# B&R Automation Studio project NAINV104C00R8L515F00 (part 35)

### Program Logical/LCS/LCSLF (IEC) - 1.00.0 - NtRecipe v5.00.0 , NtFileIO v5.00.0

#### InputRef.var
```iecst
(*2019-06-28*)
(**)
(*General*)
VAR
	p_eAct : REFERENCE TO eLCSAction;
	p_udiRstErr : REFERENCE TO UDINT;
	p_bPrep : REFERENCE TO BOOL;
	p_bEn : REFERENCE TO BOOL;
	p_bDis : REFERENCE TO BOOL;
END_VAR
(**)
(*Configuration*)
VAR
	p_tyCurrProdParam : REFERENCE TO tyProdRcpParam;
	p_bMnlAccData : REFERENCE TO BOOL;
	p_bAccData : REFERENCE TO BOOL;
	p_tyLCSProdRcpInfo : REFERENCE TO tyProdRcpParam;
	p_bChkLmtOK : REFERENCE TO BOOL;
	p_bChkLmtNG : REFERENCE TO BOOL;
	p_bAccNewRcpCond : REFERENCE TO BOOL;
	p_bUpdtNewRcpCond : REFERENCE TO BOOL;
	p_bAutoUpdtData : REFERENCE TO BOOL;
	p_bUIUpdtData : REFERENCE TO BOOL;
	p_sInfoMsg : REFERENCE TO STRING[200];
	p_sProgNm : REFERENCE TO STRING[15];
	p_bNtSettingsLoadDone : REFERENCE TO BOOL;
	p_bUIBtnSectionLdr : REFERENCE TO BOOL;
	p_bLCSSectionLeaderEn : REFERENCE TO BOOL;
	p_bMcParamSectionLdr : REFERENCE TO BOOL;
END_VAR
```

#### InputRef_Link.var
```iecst
(*2019-04-24*)
(**)
VAR
	sWidthInUMTemp : STRING[80];
	p_bLinkStartupRun : REFERENCE TO BOOL;
	p_eLinkMcParamUSCommMod : REFERENCE TO eMcSetCommMod;
END_VAR
(**)
VAR
	p_bLinkOpsRun : REFERENCE TO BOOL;
	p_bLinkMcParam : REFERENCE TO tyMcParam;
	p_bLinkConvHvBrd : REFERENCE TO BOOL;
END_VAR
```

#### Local.var
```iecst
(*2019-06-28*)
(**)
(*Local Action, State & Status*)
VAR
	eAct : eLCSAction := LCSActIdle;
	eStat : eLCSAction := LCSActIdle;
	eStatus : eFBStatus := Idle;
	udiStatus : UDINT := 0;
	sStatTxt : STRING[200] := '';
	a_sStatText : ARRAY[0..50] OF STRING[200] := ['Idling','Adding Product','Adding Multiple Products','Editing Product','Editing Multiple Products','OverWrite Product','OverWrite Multiple Products','Deleting Product','Deleting Multiple Products','Running LCS Product','Uploading Product','Uploading Multiple Products',39('')];
END_VAR
(**)
(*Local Alarm*)
VAR
	tyAlmData : tyAlmDat;
	tyInfoData : tyAlmDat;
	a_tyAlmText : ARRAY[10000..10099] OF tyAlmTxt;
END_VAR
(**)
(*Local Output*)
VAR
	udiPLCStatus : UDINT;
	bChkLmt : BOOL;
	bAccDataMnl : BOOL;
	bUpdtDataMnl : BOOL;
	sUpdtProdRcpNm : STRING[30];
	diUpdtProdWidth : DINT;
END_VAR
(**)
(*Local Input*)
VAR
	udiRstErr : UDINT := 0;
	bPrep : BOOL := TRUE;
	bEn : BOOL := TRUE;
	bDis : BOOL := FALSE;
	tyCurrProdParam : tyProdRcpParam;
	bMnlAccData : BOOL;
	bAccData : BOOL;
	tyLCSProdRcpInfo : tyProdRcpParam;
	bChkLmtOK : BOOL;
	bChkLmtNG : BOOL;
	bAccNewRcpCond : BOOL;
	bUpdtNewRcpCond : BOOL;
	bAutoUpdtData : BOOL;
	bUIUpdtData : BOOL;
	sInfoMsg : STRING[200];
	sProgNm : STRING[15] := 'LCSLF';
	bNtSettingsLoadDone : BOOL := TRUE;
END_VAR
(**)
(*Local*)
VAR
	bRstErr : BOOL;
	udiRstErrOld : UDINT;
	bInitDone : BOOL;
	bInitialDone : BOOL;
	usiStep : USINT;
	usiProdUpdtDatStep : USINT;
	udiModuleNum : UDINT := 4101;
END_VAR
```

#### Act_Action.st
```iecst
(** 2019-04-24 **)
ACTION Act_Action:

	//Reset Error
	IF (eStatus = Error) AND bRstErr THEN
		p_eAct	:= LCSActIdle;
		eStat	:= LCSActIdle;
	END_IF

	//Reset Done
	IF eStatus = Done AND p_eAct = LCSActIdle THEN
		eStat	:= LCSActIdle;
	END_IF

	//Set p_eAct
	IF eStatus = Idle THEN
		eStat	:= p_eAct;
	END_IF

END_ACTION
```

#### Act_Alarm.st
```iecst
(** 2019-04-24 **)
ACTION Act_Alarm:

	//Error
	IF EDGEPOS(eStatus = Error) THEN

		tyAlmData.sProgNm		:= p_sProgNm;
		tyAlmData.udiCode		:= udiStatus;
		tyAlmData.eSeverity		:= AlmSeverityError;
		tyAlmData.udiRunTime	:= tyAlmData.udiRunTime + 1;
		tyAlmData.bAlm			:= TRUE;
		tyAlmData.udiModuleNum  := udiModuleNum;
		g_sLCSLFProgNm			:= p_sProgNm;

		//Get Error Message
		IF tyAlmData.udiCode < 10000 OR tyAlmData.udiCode > 10099 THEN
			tyAlmData.sAlmMsg	:= 'Unknown';
			tyAlmData.sRcyMsg	:= 'Unknown';
		ELSE
			tyAlmData.sAlmMsg	:= a_tyAlmText[tyAlmData.udiCode].sAlmText;
			tyAlmData.sRcyMsg	:= a_tyAlmText[tyAlmData.udiCode].sRcyText;
		END_IF

		sStatTxt	:= tyAlmData.sAlmMsg;

	ELSIF bRstErr AND (tyAlmData.udiCode <> 0) THEN

		tyAlmData.udiCode	:= 0;
		tyAlmData.eSeverity	:= AlmSeverityNA;
		tyAlmData.sAlmMsg	:= '';
		tyAlmData.sRcyMsg	:= '';
		tyAlmData.bAlm			:= FALSE;
		sStatTxt	:= a_sStatText[eStat];

	END_IF

END_ACTION
```

#### Act_Background.st
```iecst
(** 2019-06-12 **)
ACTION Act_Background:

	//Update To Leader Recipe
	CASE usiProdUpdtDatStep OF
		0:
			//Update New Recipe Condition
			IF sUpdtProdRcpNm <> '' THEN
				IF (p_tyCurrProdParam.sRcpNm <> sUpdtProdRcpNm) THEN
					IF p_bUpdtNewRcpCond = TRUE THEN
						usiProdUpdtDatStep	:= 1;
					END_IF
				END_IF
			ELSE
				sUpdtProdRcpNm	:= p_tyCurrProdParam.sRcpNm;
				diUpdtProdWidth	:= p_tyCurrProdParam.diWidthInUM;
			END_IF

		1:
			//Manual Update Data Check
			IF p_bAutoUpdtData = FALSE THEN
				bUpdtDataMnl	:= TRUE;

				IF p_bUIUpdtData = TRUE THEN
					bUpdtDataMnl	:= FALSE;
					usiProdUpdtDatStep	:= 2;
				END_IF
			ELSE
				bUpdtDataMnl	:= FALSE;
				usiProdUpdtDatStep	:= 2;
			END_IF

		2:
			//Update New Recipe
			sUpdtProdRcpNm	:= p_tyCurrProdParam.sRcpNm;
			diUpdtProdWidth	:= p_tyCurrProdParam.diWidthInUM;

			usiProdUpdtDatStep	:= 0;

	END_CASE

END_ACTION
```

#### Act_InitGlobal.st
```iecst
(** 2019-05-07 **)
ACTION Act_InitGlobal:

	(* Always Change If Project Change *)

	//Pass Data To Link
	p_bLinkStartupRun ACCESS p_StartupRun;
	p_eLinkMcParamUSCommMod ACCESS p_McParamUSCommMod;
	p_bLinkConvHvBrd ACCESS p_OpsInvertHvBrd;

	p_bLinkOpsRun ACCESS p_OpsRun;

	//Pass Data To Internal Use
	p_eAct ACCESS p_LCS_LCSLF_LCSAct;
	p_udiRstErr ACCESS p_RstErrReset;
	p_bPrep ACCESS p_NtParamLCSLFPrep;
	p_bEn ACCESS p_McParamLCSLFEn;
	p_tyCurrProdParam ACCESS p_ProdRcpCurrRcp0;
	p_bMnlAccData ACCESS p_McParamMnlAccDat;
	p_bAccData ACCESS p_UIProdAccData;
	p_tyLCSProdRcpInfo ACCESS p_LCS_LCSLF_LCSProdRcpInfo;
	p_bChkLmtOK ACCESS p_LCSChkLmtOK;
	p_bChkLmtNG ACCESS p_LCSChkLmtNG;
	p_sProgNm ACCESS p_NtParamLCSLFProgNm;
	p_bNtSettingsLoadDone ACCESS p_StartupNtSettingsLoadDone;

	p_bUIBtnSectionLdr ACCESS P_UISectionLdr;
	p_bLCSSectionLeaderEn ACCESS p_LCSSectionLeaderEn;
	p_bMcParamSectionLdr ACCESS p_McParamSectionLeader;

	(* Always Change If Project Change *)

END_ACTION
```

#### Act_InitLocal.st
```iecst
(** 2019-06-28 **)
ACTION Act_InitLocal:

	//Input Reference Link To Local Variable
	p_eAct ACCESS ADR(eAct);
	p_udiRstErr ACCESS ADR(udiRstErr);
	p_bPrep ACCESS ADR(bPrep);
	p_bEn ACCESS ADR(bEn);
	p_bDis ACCESS ADR(bDis);
	p_tyCurrProdParam ACCESS ADR(tyCurrProdParam);
	p_bMnlAccData ACCESS ADR(bMnlAccData);
	p_bAccData ACCESS ADR(bAccData);
	p_tyLCSProdRcpInfo ACCESS ADR(tyLCSProdRcpInfo);
	p_bChkLmtOK ACCESS ADR(bChkLmtOK);
	p_bChkLmtNG ACCESS ADR(bChkLmtNG);
	p_bAccNewRcpCond ACCESS ADR(bAccNewRcpCond);
	p_bUpdtNewRcpCond ACCESS ADR(bUpdtNewRcpCond);
	p_bAutoUpdtData ACCESS ADR(bAutoUpdtData);
	p_bUIUpdtData ACCESS ADR(bUIUpdtData);
	p_sInfoMsg ACCESS ADR(sInfoMsg);
	p_sProgNm ACCESS ADR(sProgNm);
	p_bNtSettingsLoadDone ACCESS ADR(bNtSettingsLoadDone);

END_ACTION
```

#### Act_Link.st
```iecst
(** 2019-06-28 **)
ACTION Act_Link:

	p_sInfoMsg		:= 'LCS Request New Recipe';
	p_sInfoMsg		:= CONCAT(p_sInfoMsg , '$r$n');
	p_sInfoMsg		:= CONCAT(p_sInfoMsg , 'Old Recipe Name : ');
	p_sInfoMsg		:= CONCAT(p_sInfoMsg , p_tyCurrProdParam.sRcpNm);
	p_sInfoMsg		:= CONCAT(p_sInfoMsg , '$r$n');
	p_sInfoMsg		:= CONCAT(p_sInfoMsg , 'Old Recipe Width : ');
	sWidthInUMTemp	:= DINT_TO_STRING(p_tyCurrProdParam.diWidthInUM / 1000);
	p_sInfoMsg		:= CONCAT(p_sInfoMsg , sWidthInUMTemp);
	p_sInfoMsg		:= CONCAT(p_sInfoMsg , '$r$n');
	p_sInfoMsg		:= CONCAT(p_sInfoMsg , 'New Recipe Name : ');
	p_sInfoMsg		:= CONCAT(p_sInfoMsg , p_tyLCSProdRcpInfo.sRcpNm);
	p_sInfoMsg		:= CONCAT(p_sInfoMsg , '$r$n');
	p_sInfoMsg		:= CONCAT(p_sInfoMsg , 'New Recipe Width : ');
	sWidthInUMTemp	:= DINT_TO_STRING(p_tyLCSProdRcpInfo.diWidthInUM / 1000);
	p_sInfoMsg		:= CONCAT(p_sInfoMsg , sWidthInUMTemp);

	//Accept New Recipe Condition
	p_bAccNewRcpCond	:= p_bLinkOpsRun = TRUE AND p_bLinkConvHvBrd = FALSE;

END_ACTION
```

#### Act_LinkAction.st
```iecst
(** 2019-04-24 **)
ACTION Act_LinkAction:

END_ACTION
```

#### Act_LinkEn.st
```iecst
(** 2019-04-24 **)
ACTION Act_LinkEn:

	//Link bPrep, bEn & bDis
	p_bDis	:= (p_bLinkStartupRun = TRUE) OR (p_eLinkMcParamUSCommMod = McSetCommModHermes);

END_ACTION
```

#### Act_Main.st
```iecst
(** 2019-06-28 **)
ACTION Act_Main:

	//Main
	CASE eStat OF

		LCSActIdle:
			IF eStatus <> Idle THEN	//Reset Data
				//Private
				usiStep		:= 0;
				bAccDataMnl	:= FALSE;
				bChkLmt		:= FALSE;

				tyInfoData.sProgNm		:= '';
				tyInfoData.udiCode		:= 0;
				tyInfoData.eSeverity	:= AlmSeverityNA;
				tyInfoData.sAlmMsg		:= '';

				sStatTxt	:= a_sStatText[eStat];

			END_IF

			eStatus			:= Idle;
			udiPLCStatus	:= 65534;

		LCSActRunProd:
			IF eStatus = Idle OR eStatus = Busy THEN

				eStatus			:= Busy;
				udiPLCStatus	:= 65535;

				sStatTxt	:= a_sStatText[eStat];

				CASE usiStep OF
					0:
						//Check Limit
						bChkLmt	:= TRUE;

						IF p_bChkLmtOK = TRUE THEN
							usiStep			:= 1;
						ELSIF p_bChkLmtNG = TRUE THEN
							eStatus			:= Done;
							udiPLCStatus	:= 10010;	//Out Of Range While Accepting New Recipe
						END_IF

					1:
						//Manual Accept Data Check
						IF p_bMnlAccData = TRUE THEN
							bAccDataMnl	:= TRUE;

							//Info Message
							tyInfoData.sProgNm		:= p_sProgNm;
							tyInfoData.udiCode		:= 10000;
							tyInfoData.eSeverity	:= AlmSeverityInfo;
							tyInfoData.sAlmMsg		:= p_sInfoMsg;

							IF p_bAccData = TRUE THEN
								p_bAccData 	:= FALSE; // 2023_07_06_Debug for Manual Accept Data automatically accept after product change many times
								bAccDataMnl	:= FALSE;
								usiStep		:= 2;
							END_IF
						ELSE
							bAccDataMnl	:= FALSE;
							p_bAccData	:= FALSE; // 2023_07_06_Debug for Manual Accept Data automatically accept after product change many times
							usiStep		:= 2;
						END_IF

					2:
						//Accept New Recipe Condition
						IF p_bAccNewRcpCond = TRUE THEN
							usiStep	:= 3;
						ELSE
							//Info Message
							tyInfoData.sProgNm		:= p_sProgNm;
							tyInfoData.udiCode		:= 10000;
							tyInfoData.eSeverity	:= AlmSeverityInfo;
							tyInfoData.sAlmMsg		:= p_sInfoMsg;
						END_IF

					3:
						//Accept New Recipe
						p_tyCurrProdParam	:= p_tyLCSProdRcpInfo;

						IF p_bLCSSectionLeaderEn = TRUE THEN
							p_bMcParamSectionLdr	:= TRUE;
							p_bUIBtnSectionLdr		:= TRUE;
						ELSE
							p_bMcParamSectionLdr	:= FALSE;
							p_bUIBtnSectionLdr		:= FALSE;

						END_IF

						usiStep	:= 4;

					4:
						//Clear Info Message
						tyInfoData.sProgNm		:= '';
						tyInfoData.udiCode		:= 0;
						tyInfoData.eSeverity	:= AlmSeverityNA;
						tyInfoData.sAlmMsg		:= '';

						usiStep	:= 0;

						eStatus			:= Done;
						udiPLCStatus	:= 0;

				END_CASE

			END_IF

		ELSE
			IF eStatus = Idle OR eStatus = Busy THEN
				eStatus	:= Done;
			END_IF

	END_CASE

END_ACTION
```

#### Act_Main_Disable.st
```iecst
(** 2019-06-12 **)
ACTION Act_Main_Disable:

	usiProdUpdtDatStep		:= 0;

END_ACTION
```

#### Act_RstErr.st
```iecst
(** 2019-04-24 **)
ACTION Act_RstErr:

	IF p_udiRstErr <> udiRstErrOld THEN
		bRstErr			:= TRUE;
		udiRstErrOld	:= p_udiRstErr;
	ELSE
		bRstErr			:= FALSE;
	END_IF

END_ACTION
```

#### Cyclic.st
```iecst
(** 2019-04-24 **)
PROGRAM _CYCLIC

	IF bInitDone = FALSE THEN
		bInitDone	:= TRUE;

		Act_InitLocal;
		Act_InitGlobal;

	ELSIF bInitialDone = FALSE THEN
		IF p_bNtSettingsLoadDone = TRUE THEN
			bInitialDone	:= TRUE;

			Act_Initial;
		END_IF

	ELSE

		Act_RstErr;
		Act_LinkAction;
		Act_Action;
		Act_LinkEn;

		IF (p_bPrep = TRUE) AND (p_bEn = TRUE) AND (p_bDis = FALSE) THEN
			Act_Link;
			Act_Background;
			Act_Main;

		ELSE
			Act_Main_Disable;

			IF eStat <> LCSActIdle THEN
				eStatus			:= Done;
				udiPLCStatus	:= 10002;	//LCS Leader Follower Disabled
			ELSE
				eStatus	:= Idle;
			END_IF
		END_IF

		Act_Alarm;

	END_IF

END_PROGRAM
```

#### Init.st
```iecst
(** 2019-06-12 **)
PROGRAM _INIT

	(* Always Change If Project Change *)

	//Pass Address To Global Address For External Use
	//Action, State & Status
	p_LCSLFStat		:= ADR(eStat);
	p_LCSLFStatus	:= ADR(eStatus);
	p_LCSLFStatTxt	:= ADR(sStatTxt);

	//Alarm
	p_LCSLFAlmData	:= ADR(tyAlmData);
	p_LCSLFInfoData	:= ADR(tyInfoData);

	//Output
	p_LCSLF_PLCStatus		:= ADR(udiPLCStatus);
	p_LCSLFChkLmt			:= ADR(bChkLmt);
	p_LCSLFAccDataMnl		:= ADR(bAccDataMnl);
	p_LCSLFUpdtDataMnl		:= ADR(bUpdtDataMnl);
	p_LCSLFUpdtProdRcpNm	:= ADR(sUpdtProdRcpNm);
	p_LCSLFUpdtProdWidth	:= ADR(diUpdtProdWidth);

	(* Always Change If Project Change *)

END_PROGRAM
```

### Ops.typ - Do Not Change!!!
```iecst
(*2019-04-16*)
(**)

TYPE
	eOperationsAction :
		(
		OperationsActIdle,
		OperationsActStart,
		OperationsActStop,
		OperationsActStep,
		OperationsActError
		);
END_TYPE

(**)

TYPE
	eOperationsStatus :
		(
		OperationsStatusRun,
		OperationsStatusStop,
		OperationsStatusCycleStopping,
		OperationsStatusStep
		);
END_TYPE
```

### Ops.var - Change By Project
```iecst
(*2019-04-16*)
(**)
(*Action & State & Status*)
VAR
	p_OpsStat : UDINT;
	p_OpsStatus : UDINT;
	p_OpsStatTxt : UDINT;
END_VAR
(**)
(*Alarm*)
(**)
(*Output*)
VAR
	p_OpsOpsStatus : UDINT;
	p_OpsStatusRun : UDINT;
	p_OpsStatusStop : UDINT;
	p_OpsStatusCycleStop : UDINT;
	p_OpsStatusStep : UDINT;
	p_OpsRun : UDINT;
	p_OpsStop : UDINT;
	p_OpsStep : UDINT;
END_VAR
```

### Program Logical/Operations/Ops (IEC, version 1.00.0) - 1.00.0 - 

#### Init.st - Change By Project
```iecst
(** 2019-04-16 **)
PROGRAM _INIT

	(* Always Change If Project Change *)

	//Pass Address To Global Address For External Use
	//Action, State & Status
	p_OpsStat		:= ADR(eStat);
	p_OpsStatus		:= ADR(eStatus);
	p_OpsStatTxt	:= ADR(sStatTxt);

	//Alarm

	//Output
	p_OpsOpsStatus			:= ADR(eOpsStatus);
	p_OpsStatusRun			:= ADR(bStatusRun);
	p_OpsStatusStop			:= ADR(bStatusStop);
	p_OpsStatusCycleStop	:= ADR(bStatusCycleStop);
	p_OpsStatusStep			:= ADR(bStatusStep);
	p_OpsRun				:= ADR(bRun);
	p_OpsStop				:= ADR(bStop);
	p_OpsStep				:= ADR(bStep);

	(* Always Change If Project Change *)

END_PROGRAM
```

#### Act_InitGlobal.st - Change By Project
```iecst
(** 2019-03-22 **)
ACTION Act_InitGlobal:

	(* Always Change If Project Change *)

	//Pass Data To Link
	p_bOpsInvertPaused ACCESS p_OpsInvertPaused;

	//Pass Data To Internal Use
	p_eAct ACCESS p_UIOpsAct;
	p_udiRstErr ACCESS p_RstErrReset;
	p_bNtSettingsLoadDone ACCESS p_StartupNtSettingsLoadDone;

	(* Always Change If Project Change *)

END_ACTION
```

#### InputRef_Link.var - Change By Project
```iecst
(*2019-01-20*)
(**)
VAR
	p_bOpsInvertPaused : REFERENCE TO BOOL;
END_VAR
```

#### Act_Link.st - Change By Project
```iecst
(** 2019-01-20 **)
ACTION Act_Link:

	p_bPaused	:=  p_bOpsInvertPaused;

END_ACTION
```

#### Cyclic.st - Do Not Change!!!
```iecst
(** 2019-03-29 **)
PROGRAM _CYCLIC

	IF bInitDone = FALSE THEN
		bInitDone	:= TRUE;

		Act_InitLocal;
		Act_InitGlobal;

	ELSIF bInitialDone = FALSE THEN
		IF p_bNtSettingsLoadDone = TRUE THEN
			bInitialDone	:= TRUE;

			Act_Initial;
		END_IF

	ELSE

		Act_RstErr;
		Act_LinkAction;
		Act_Action;
		Act_Link;
		Act_Main;

	END_IF

END_PROGRAM
```

#### Act_Action.st - Do Not Change!!!
```iecst
(** 2019-03-25 **)
ACTION Act_Action:

	//Reset Error
	IF (eStatus = Error) AND bRstErr THEN
		p_eAct	:= OperationsActIdle;
		eStat	:= OperationsActIdle;
	END_IF

	//Set p_eAct
	IF eStatus = Idle OR eStatus = Busy OR eStatus = Done THEN
		eStat	:= p_eAct;
	END_IF

END_ACTION
```

#### Act_Main.st - Do Not Change!!!
```iecst
(** 2019-04-16 **)
ACTION Act_Main:

	IF eStatOld <> eStat THEN
		usiStep		:= 0;

		sStatTxt	:= a_sStatText[eStat];

		eStatOld	:= eStat;

		eStatus		:= Busy;
	END_IF

	//Main
	CASE eStat OF

		OperationsActIdle:
			eStatus	:= Idle;

		OperationsActStart:
			IF eStatus = Idle OR eStatus = Busy THEN

				eOpsStatus			:= OperationsStatusRun;
				bStatusRun			:= TRUE;
				bStatusStop			:= FALSE;
				bStatusCycleStop	:= FALSE;
				bStatusStep			:= FALSE;

				bRun		:= TRUE;
				bStop		:= FALSE;
				bStep		:= FALSE;

				eStatus	:= Done;

			END_IF

		OperationsActStop:
			IF eStatus = Idle OR eStatus = Busy THEN

				eStatus	:= Busy;

				eOpsStatus			:= OperationsStatusCycleStopping;
				bStatusRun			:= FALSE;
				bStatusStop			:= FALSE;
				bStatusCycleStop	:= TRUE;
				bStatusStep			:= FALSE;

				bStop	:= TRUE;

				IF p_bPaused THEN

					bRun	:= FALSE;

					eOpsStatus			:= OperationsStatusStop;
					bStatusRun			:= FALSE;
					bStatusStop			:= TRUE;
					bStatusCycleStop	:= FALSE;
					bStatusStep			:= FALSE;

					eStatus	:= Done;

				END_IF

			END_IF

		OperationsActStep:
			IF eStatus = Idle OR eStatus = Busy THEN

				eStatus	:= Busy;

				eOpsStatus			:= OperationsStatusStep;
				bStatusRun			:= FALSE;
				bStatusStop			:= FALSE;
				bStatusCycleStop	:= FALSE;
				bStatusStep			:= TRUE;

				bRun	:= TRUE;

				CASE usiStep OF

					0:
						bStep	:= FALSE;
						usiStep	:= 1;

					1:
						bStep	:= TRUE;

				END_CASE

				IF p_bPaused THEN
					eStatus	:= Done;
				END_IF

			END_IF

		OperationsActError:
			IF eStatus = Idle OR eStatus = Busy THEN

				eOpsStatus			:= OperationsStatusStop;
				bStatusRun			:= FALSE;
				bStatusStop			:= TRUE;
				bStatusCycleStop	:= FALSE;
				bStatusStep			:= FALSE;

				bRun		:= FALSE;
				bStop		:= FALSE;
				bStep		:= FALSE;

				eStatus	:= Done;

			END_IF

	END_CASE

END_ACTION
```

#### InputRef.var - Do Not Change!!!
```iecst
(*2019-03-25*)
(**)
(*General*)
VAR
	p_eAct : REFERENCE TO eOperationsAction;
	p_udiRstErr : REFERENCE TO UDINT;
	p_bPaused : REFERENCE TO BOOL;
	p_bNtSettingsLoadDone : REFERENCE TO BOOL;
END_VAR
```

#### Local.var - Do Not Change!!!
```iecst
(*2019-04-30*)
(**)
(*Local Action, State & Status*)
VAR
	eAct : eOperationsAction := OperationsActIdle;
	eStat : eOperationsAction := OperationsActIdle;
	eStatus : eFBStatus := Idle;
	sStatTxt : STRING[200] := '';
	a_sStatText : ARRAY[0..50] OF STRING[200] := ['Idling','Starting Operations','Sequence Stopping Operations','Pause Operations In Step','Accepting New Data','Accepted New Data','Error Immediate Stop Operations',44('')];
END_VAR
(**)
(*Local Alarm*)
(**)
(*Local Output*)
VAR
	eOpsStatus : eOperationsStatus := OperationsStatusStop;
	bStatusRun : BOOL;
	bStatusStop : BOOL := TRUE;
	bStatusCycleStop : BOOL;
	bStatusStep : BOOL;
	bRun : BOOL;
	bStop : BOOL;
	bStep : BOOL;
END_VAR
(**)
(*Local Input*)
VAR
	udiRstErr : UDINT := 0;
	bPaused : BOOL;
	bNtSettingsLoadDone : BOOL := TRUE;
END_VAR
(**)
(*Local*)
VAR
	bRstErr : BOOL;
	udiRstErrOld : UDINT;
	bInitDone : BOOL;
	bInitialDone : BOOL;
	eStatOld : eOperationsAction := OperationsActIdle;
	usiStep : USINT;
END_VAR
```

### OpsInvert.var - Change By Project
```iecst
(*2020-10-06*)
(**)
(*Action & State & Status*)
(**)
(*Alarm*)
VAR
	p_OpsInvertAlmData : UDINT;
	p_OpsInvertAlmData1 : UDINT;
END_VAR
(**)
(*Output*)
VAR
	p_OpsInvertStepTxt : UDINT;
	p_OpsInvertPaused : UDINT;
	p_OpsInvertHvBrd : UDINT;
	p_OpsInvertGdBrd : UDINT;
END_VAR
(**)
VAR
	p_OpsInvertStepInitConv : UDINT;
	p_OpsInvertStepInitAwayStpr : UDINT;
	p_OpsInvertStepInitTwdStpr : UDINT;
	p_OpsInvertStepInitDone : UDINT;
	p_OpsInvertStepUSStandby : UDINT;
	p_OpsInvertStepUSCommTmr : UDINT;
	p_OpsInvertStepEntToEnd : UDINT;
	p_OpsInvertStepEntToInOff : UDINT;
	p_OpsInvertStepRev : UDINT;
	p_OpsInvertStepPreExit : UDINT;
	p_OpsInvertStepDSStandby : UDINT;
	p_OpsInvertStepDSCommTmr : UDINT;
	p_OpsInvertStepExitBrd : UDINT;
	p_OpsInvertStepInvert : UDINT;
END_VAR
(* *)
VAR
	p_OpsInvertStepAWMove : UDINT;
	p_OpsInvertStepOpsSafeMode : UDINT;
END_VAR
(**)
VAR
	p_OpsInvertBrdInserted : UDINT;
	p_OpsInvertBrdRemoved : UDINT;
END_VAR
(**)
VAR
	p_OpsInvertUSSMEMAAct : UDINT;
	p_OpsInvertDSSMEMAAct : UDINT;
	p_OpsInvertConvAct : UDINT;
	p_OpsInvertStopperAct : UDINT;
	p_OpsInvertInvertAct : UDINT;
	p_OpsInvertAWAct : UDINT;
	p_OpsInvertClampAct : UDINT;
	p_OpsInvertInletShutterAct : UDINT;
	p_OpsInvertOutletShutterAct : UDINT;
	p_OpsInvertClamp1Act : UDINT;
	p_OpsInvertClamp2Act : UDINT;
	p_OpsInvertClamp3Act : UDINT;
END_VAR
(**)
VAR
	p_OpsInvertUSSMEMA2Act : UDINT;
	p_OpsInvertOnceTwicePCBOut : UDINT;
	p_OpsInvertStepInvRtrnUSStandby : UDINT;
	p_OpsInvertStepInvRtrnUSCommTmr : UDINT;
	p_OpsInvertStepInvRtrnEntToEnd : UDINT;
	p_OpsInvertStepInvRtrnEntToInOff : UDINT;
END_VAR
(**)
VAR
	p_OpsInvertInvertCurrPos : UDINT;
END_VAR
```

### OpsInvert.typ - Do Not Change!!!
```iecst
(*2020-10-08*)
(**)
(*Sequence*)

TYPE
	eInvertStep :
		(
		InvertStepNA,
		InvertStepInitChkCondition,
		InvertStepInitInvertComplChk,
		InvertStepInitClampUnblk,
		InvertStepInitConvAwayLftSen,
		InvertStepInitConvAwayRgtSen,
		InvertStepInitStopperBlk,
		InvertStepInitConvTwdLftSen,
		InvertStepInitConvTwdRgtSen,
		InvertStepInitStopperUnblk,
		InvertStepInitConvToRgt,
		InvertStepInitInvRtrnConv,
		InvertStepInitShuttersInOutClose,
		InvertStepChkCondition,
		InvertStepShuttersInOutClose,
		InvertStepAWMov,
		InvertStepSafetyInOutClose,
		InvertStepShutterCloseWaitForSig,
		InvertStepChkShutterCond,
		InvertStepShuttersInOutOpen,
		InvertStepShuttersInOpenOutClose,
		InvertStepStopperPosChk,
		InvertStepStopperBlk,
		InvertStepStopperUnblk,
		InvertStepUSStandby,
		InvertStepUSTmr,
		InvertStepUSCommTmr,
		InvertStepEntToEnd,
		InvertStepEntToInOff,
		InvertStepStopperBlkAftEnt,
		InvertStepRev,
		InvertStepShuttersInClose,
		InvertStepInvertComplChk,
		InvertStepClampBlkBefInvert,
		InvertStepShuttersCloseBefInvert,
		InvertStepInvert,
		InvertStepInvalidPosRecoverBrd,
		InvertStepClampUnblkAftInvert,
		InvertStepStopperUnblkAftInvert,
		InvertStepPreExit,
		InvertStepDSInOutletShutterOpen,
		InvertStepOutletShutterOpen,
		InvertStepDSStandby,
		InvertStepDSTmr,
		InvertStepDSCommTmr,
		InvertShuttersInOutCloseBefInitR,
		InvertShuttersInOutCloseBefInit,
		InvertStepExitBrd,
		InvertStepPCBOut,
		InvertStepInvRtrnUSStandby,
		InvertStepInvRtrnUSTmr,
		InvertStepInvRtrnUSCommTmr,
		InvertStepInvRtrnEntToEnd,
		InvertStepInvRtrnEntToInOff,
		InvertStepShuttersInCloseOutOpen
		);
END_TYPE

(**)

TYPE
	eInvertPos :
		(
		InvertCurrPosAtRemote,
		InvertCurrPosAtHome,
		InvertPosInvalid
		);
END_TYPE
```

### Program Logical/Operations/OpsInvert (IEC, version 1.00.0) - 1.00.0 - 

#### Init.st - Change By Project
```iecst
(** 2020-10-09 **)
PROGRAM _INIT

	(* Always Change If Project Change *)

	//Pass Address To Global Address For External Use
	//Action, State & Status

	//Alarm
	p_OpsInvertAlmData	:= ADR(tyAlmData);
	p_OpsInvertAlmData1	:= ADR(tyAlmData1);

	//Output
	p_OpsInvertStepTxt		:= ADR(sStepTxt);
	p_OpsInvertPaused		:= ADR(bPaused);
	p_OpsInvertGdBrd 		:= ADR(bGdBrd);
	p_OpsInvertHvBrd		:= ADR(bHvBrd);

	p_OpsInvertUSSMEMAAct	:= ADR(eUSSMEMAAct);
	p_OpsInvertDSSMEMAAct	:= ADR(eDSSMEMAAct);
	p_OpsInvertConvAct		:= ADR(eConvAct);
	p_OpsInvertStopperAct	:= ADR(eStopperAct);
	p_OpsInvertInvertAct	:= ADR(eInvertAct);
	p_OpsInvertAWAct		:= ADR(eAWAct);
	p_OpsInvertClampAct		:= ADR(eClampAct);
	p_OpsInvertInletShutterAct	:= ADR(eInletShutterAct);
	p_OpsInvertOutletShutterAct	:= ADR(eOutletShutterAct);
	p_OpsInvertClamp1Act		:= ADR(eClamp1Act);
	p_OpsInvertClamp2Act		:= ADR(eClamp2Act);
	p_OpsInvertClamp3Act		:= ADR(eClamp3Act);

	p_OpsInvertStepInitConv			:= ADR(bStepInitConv);
	p_OpsInvertStepInitAwayStpr		:= ADR(bStepInitAwayStopper);
	p_OpsInvertStepInitTwdStpr		:= ADR(bStepInitTwdStopper);
	p_OpsInvertStepInitDone			:= ADR(bStepInitDone);
	p_OpsInvertStepUSStandby		:= ADR(bStepUSStandby);
	p_OpsInvertStepUSCommTmr		:= ADR(bStepUSCommTmr);
	p_OpsInvertStepEntToEnd			:= ADR(bStepEntToEnd);
	p_OpsInvertStepEntToInOff		:= ADR(bStepEntToInOff);
	p_OpsInvertStepRev				:= ADR(bStepRev);
	p_OpsInvertStepPreExit			:= ADR(bStepPreExit);
	p_OpsInvertStepDSStandby		:= ADR(bStepDSStandby);
	p_OpsInvertStepDSCommTmr		:= ADR(bStepDSCommTmr);
	p_OpsInvertStepExitBrd			:= ADR(bStepExitBrd);
	p_OpsInvertStepInvert			:= ADR(bStepInvert);
	p_OpsInvertStepAWMove			:= ADR(bStepAWMov);
	p_OpsInvertStepOpsSafeMode		:= ADR(bStepSafeMode);

	p_OpsInvertBrdInserted			:= ADR(bBrdInserted);
	p_OpsInvertBrdRemoved			:= ADR(bBrdRemoved);

	p_OpsInvertInvertCurrPos		:= ADR(eInvertCurrPos);

	p_OpsInvertUSSMEMA2Act				:= ADR(eUSSMEMA2Act);
	p_OpsInvertOnceTwicePCBOut			:= ADR(bInvOnceTwicePCBOut);
	p_OpsInvertStepInvRtrnUSStandby		:= ADR(bStepInvRtrnUSStandby);
	p_OpsInvertStepInvRtrnUSCommTmr		:= ADR(bStepInvRtrnUSCommTmr);
	p_OpsInvertStepInvRtrnEntToEnd		:= ADR(bStepInvRtrnEntToEnd);
	p_OpsInvertStepInvRtrnEntToInOff	:= ADR(bStepInvRtrnEntToInOff);

	(* Always Change If Project Change *)

END_PROGRAM
```

#### Act_InitGlobal.st - Change By Project
```iecst
(** 2020-10-06 **)
ACTION Act_InitGlobal:

	(* Always Change If Project Change *)

	//Pass Data To Link
	p_usiLinkProdRcpCurrRcpMcMod ACCESS p_ProdRcpCurrRcp1McMod;
	p_bLinkConvHvBrd ACCESS p_ConvHvBrd;

	p_bLinkInvertHomeSen ACCESS p_DIInvertHomeSen;
	p_bLinkInvertRemoteSen ACCESS p_DIInvertRemoteSen;

	p_bLinkUSHermesBlkUS ACCESS p_USHermesBlkUS;
	p_bLinkUSHermes2BlkUS ACCESS p_USHermes2BlkUS;
	p_bLinkFollower1USAllow ACCESS p_Follower1USAllow;
	p_bLinkFollower1DSAllow ACCESS p_Follower1DSAllow;
	p_bLinkLFFollowerUSAllow ACCESS p_LFFollowerUSAllow;
	p_bLinkLFFollowerDSAllow ACCESS p_LFFollowerDSAllow;

	p_bLinkFollower1WaitRlsBrd ACCESS p_Follower1WaitRlsBrd;

	p_diFwdDlyTm ACCESS p_NtParamConvFwdDlyTm;
	p_diRevDlyTm ACCESS p_NtParamConvRevDlyTm;

	p_bLinkUIRtnBrdReset ACCESS p_UIRtnBrdReset;
	p_bLinkUIRtnBrdResetBtn ACCESS p_UIRtnBrdResetBtn;

	//Pass Data To Internal Use
	p_udiRstErr ACCESS p_RstErrReset;
	p_bRun ACCESS p_OpsRun;
	p_bStop ACCESS p_OpsStop;
	p_bStep ACCESS p_OpsStep;

	p_eConvDirection ACCESS p_NtParamProjConvDir;
	p_eUSCommMod ACCESS p_McParamUSCommMod;
	p_eDSCommMod ACCESS p_McParamDSCommMod;

	p_eUSSMEMAStat ACCESS p_USSMEMAStat;
	p_eUSSMEMAStatus ACCESS p_USSMEMAStatus;
	p_bUSSMEMATransporting ACCESS p_USSMEMATransporting;
	p_bUSSMEMAConvStart ACCESS p_USSMEMAConvStart;
	p_bUSSMEMAConvStop ACCESS p_USSMEMAConvStop;
	p_bUSSMEMAUSRdy ACCESS p_USSMEMAUSRdy;
	p_bUSSMEMAUSGdBrdRdy ACCESS p_USSMEMAUSGdBrdRdy;

	p_eDSSMEMAStat ACCESS p_DSSMEMAStat;
	p_eDSSMEMAStatus ACCESS p_DSSMEMAStatus;
	p_bDSSMEMAConvStart ACCESS p_DSSMEMAConvStart;
	p_bDSSMEMAConvStop ACCESS p_DSSMEMAConvStop;
	p_bDSSMEMATimer ACCESS p_DSSMEMATimer;

	p_bUSHermesTransporting ACCESS p_USHermesTransporting;
	p_bUSHermesStopTransport ACCESS p_USHermesStopTransport;

	p_bUSHermesUSRdy ACCESS p_USHermesUSRdy;
	p_bUSHermesUSGdRdy ACCESS p_USHermesUSGdRdy;

	p_bDSHermesTransporting ACCESS p_DSHermesTransporting;
	p_bDSHermesStopTransport ACCESS p_DSHermesStopTransport;

	p_eConvStat ACCESS p_ConvStat;
	p_eConvStatus ACCESS p_ConvStatus;
	p_bConvHvBrd ACCESS p_ConvHvBrd;

	p_eStopperStat ACCESS p_PneuNoSenStopperStat;
	p_eStopperStatus ACCESS p_PneuNoSenStopperStatus;
	p_bStopperExtended ACCESS p_PneuNoSenStopperExtended;
	p_bStopperRetracted ACCESS p_PneuNoSenStopperRetracted;

	p_eClampStat ACCESS p_PneuNoSenClampStat;
	p_eClampStatus ACCESS p_PneuNoSenClampStatus;

	p_eInvertStat ACCESS p_MotorBrkStat;
	p_eInvertStatus ACCESS p_MotorBrkStatus;

	p_eInletShutterStat ACCESS p_Pneu2SenInShutterStat;
	p_eInletShutterStatus ACCESS p_Pneu2SenInShutterStatus;
	p_bInletShutterOpen ACCESS p_DIInShutterOpenRS;
	p_bInletShutterClose ACCESS p_DIInShutterCloseRS;

	p_eOutletShutterStat ACCESS p_Pneu2SenOutShutterStat;
	p_eOutletShutterStatus ACCESS p_Pneu2SenOutShutterStatus;
	p_bOutletShutterOpen ACCESS p_DIOutShutterOpenRS;
	p_bOutletShutterClose ACCESS p_DIOutShutterCloseRS;

	p_eClamp1Stat ACCESS p_Pneu2SenClamp1Stat;
	p_eClamp1Status ACCESS p_Pneu2SenClamp1Status;
	p_bClampRS1 ACCESS p_DIClampRS1;
	p_bUnClampRS1 ACCESS p_DIUnClampRS1;

	p_eClamp2Stat ACCESS p_Pneu2SenClamp2Stat;
	p_eClamp2Status ACCESS p_Pneu2SenClamp2Status;
	p_bClampRS2 ACCESS p_DIClampRS2;
	p_bUnClampRS2 ACCESS p_DIUnClampRS2;

	p_eClamp3Stat ACCESS p_Pneu2SenClamp3Stat;
	p_eClamp3Status ACCESS p_Pneu2SenClamp3Status;
	p_bClampRS3 ACCESS p_DIClampRS3;
	p_bUnClampRS3 ACCESS p_DIUnClampRS3;

	p_bLeftSen ACCESS p_DIConvLftSen;
	p_bRightSen ACCESS p_DIConvRgtSen;

	p_bClamp2Sen ACCESS p_DIClamp2Sen;
	p_bClamp3Sen ACCESS p_DIClamp3Sen;

	p_eAWStat ACCESS p_AWOpenStat;
	p_eAWStatus ACCESS p_AWOpenStatus;
	p_bAWWidthPosDiff ACCESS p_AWOpenWidthPosDiff;

	p_sProgNm ACCESS p_NtParamOpsConvProgNm;
	p_bNtSettingsLoadDone ACCESS p_StartupNtSettingsLoadDone;

	p_bClampDis ACCESS p_McParamClampDis;
	p_bClampPrep ACCESS p_NtParamProjClampPrep;
	p_eClampOption ACCESS p_NtParamProjClampOption;

	p_bInletShutterPrep ACCESS p_NtParamProjInletShutPrep;
	p_bInletShutterDis ACCESS p_McParamInShutterDis;
	p_bOutletShutterPrep ACCESS p_NtParamProjOutletShutPrep;
	p_bOutletShutterDis ACCESS p_McParamOutShutterDis;

	// Nutek Param
	p_bDBAOnRgtSen ACCESS p_NtParamProjDBAOnRgtSen;

	p_bMachineSafetyPrep ACCESS p_NTParamMachineSafetySig; 		// ADD
	p_bUnlockCovPrep ACCESS p_NTParamUnlockCovPrep;			  	// ADD
	p_bLinkDICoverSwitchSig2 ACCESS p_DICoverSWSig2;			// ADD
	p_bLinkUIBypsCoverSWPress1 ACCESS p_UIBypassTopCover1;		// ADD

	p_bLinkDIUnlockCoverSigFromDS ACCESS p_DIUnlockCoverSigFromDS;		// ADD
	p_bLinkDIUnlockCoverSigFromUS ACCESS p_DIUnlockCoverSigFromUS;		// ADD
	p_bLinkDISafetySigFromDS ACCESS p_DIUnlockSafetySigFromDS;
	p_bLinkDISafetySigFromUS ACCESS p_DIUnlockSafetySigFromUS;

	//InvertOnce & InvertTwice_2023_0032B01
	p_eUSComm2Mod ACCESS p_McParamUSComm2Mod;
	p_eUSSMEMA2Stat ACCESS p_USSMEMA2Stat;
	p_eUSSMEMA2Status ACCESS p_USSMEMA2Status;
	p_bUSSMEMA2Transporting ACCESS p_USSMEMA2Transporting;
	p_bUSSMEMA2ConvStart ACCESS p_USSMEMA2ConvStart;
	p_bUSSMEMA2ConvStop ACCESS p_USSMEMA2ConvStop;
	p_bUSSMEMA2USRdy ACCESS p_USSMEMA2USRdy;
	p_bUSSMEMA2USGdBrdRdy ACCESS p_USSMEMA2USGdBrdRdy;

	//Hermes Action & Route
	p_iHermesAction ACCESS p_USHermesAction;
	p_bUSReversal ACCESS p_HermesSwitchtoReverseTransport;//p_USHermes2SwitchtoReverseRcv;
	p_bHermesEntToReversePosition ACCESS p_HermesEntToReversePosition;

//	p_bUSHermesUSRdy ACCESS p_USHermesUSRdy;
//	p_bUSHermesUSGdRdy ACCESS p_USHermesUSGdRdy;
//	p_bDSReversal ACCESS
	(* Always Change If Project Change *)

END_ACTION
```

#### InputRef_Link.var - Change By Project
```iecst
(*2018-12-11*)
(**)
(*External Data*)
VAR
	p_usiLinkProdRcpCurrRcpMcMod : REFERENCE TO USINT;
	p_bLinkConvHvBrd : REFERENCE TO BOOL;
	p_bLinkInvertHomeSen : REFERENCE TO BOOL;
	p_bLinkInvertRemoteSen : REFERENCE TO BOOL;
END_VAR
(**)
VAR RETAIN
	eInvertReqPos : eInvertPos;
END_VAR
VAR
	eInvertCurrPos : eInvertPos;
	bInvertCompl : BOOL;
END_VAR
(**)
VAR
	p_bLinkUSHermesBlkUS : REFERENCE TO BOOL;
	p_bLinkUSHermes2BlkUS : REFERENCE TO BOOL;
	p_bLinkLFFollowerUSAllow : REFERENCE TO BOOL;
	p_bLinkLFFollowerDSAllow : REFERENCE TO BOOL;
	p_bLinkFollower1USAllow : REFERENCE TO BOOL;
	p_bLinkFollower1DSAllow : REFERENCE TO BOOL;
	p_bLinkFollower1WaitRlsBrd : REFERENCE TO BOOL;
END_VAR
(**)
VAR
	p_bLinkUIRtnBrdReset : REFERENCE TO BOOL;
	p_bLinkUIRtnBrdResetBtn : REFERENCE TO BOOL;
END_VAR
(**)
VAR
	p_diFwdDlyTm : REFERENCE TO DINT;
	p_diRevDlyTm : REFERENCE TO DINT;
END_VAR
```

#### Act_LinkEn.st - Change By Project
```iecst
(** 2019-01-11 **)
ACTION Act_LinkEn:

END_ACTION
```

#### Act_Link.st - Change By Project
```iecst
(** 2018-12-11 **)
ACTION Act_Link:
	//test
	p_bAWWidthPosDiff ACCESS ADR(btest);
	// ADD Go to Standby
	p_bGoToStandby	:= (p_bLinkUIBypsCoverSWPress1 AND p_bUnlockCovPrep) OR ((p_bLinkDIUnlockCoverSigFromDS = TRUE OR p_bLinkDIUnlockCoverSigFromUS = TRUE) AND p_bMachineSafetyPrep) ;

	IF p_bRun = TRUE AND EDGEPOS(p_bLinkDICoverSwitchSig2) THEN	// ADD
		eGotoOpsStep	:=	InvertStepInitChkCondition;
	END_IF

	//Upstream Allow
	p_bUSAllow		:= p_bLinkFollower1USAllow AND (p_bLinkUSHermesBlkUS = FALSE OR p_bLinkUSHermes2BlkUS = FALSE) AND p_bLinkLFFollowerUSAllow AND (p_bGoToStandby = FALSE);

	p_bRtrnUSAllow	:= p_bLinkFollower1USAllow AND p_bLinkUSHermesBlkUS = FALSE AND p_bLinkLFFollowerUSAllow AND (p_bGoToStandby = FALSE) AND (p_bLinkUIRtnBrdResetBtn = FALSE AND p_bLinkUIRtnBrdReset = FALSE);

	//Downstream Allow
	p_bDSAllow		:= p_bLinkFollower1DSAllow AND (NOT p_bLinkFollower1WaitRlsBrd)AND p_bLinkLFFollowerDSAllow;

	p_bRtrnDSAllow 	:= p_bLinkFollower1DSAllow AND (NOT p_bLinkFollower1WaitRlsBrd)AND p_bLinkLFFollowerDSAllow;

	//Update Request Invert Position
	IF p_usiLinkProdRcpCurrRcpMcMod = 0 THEN
		IF eInvertCurrPos <> InvertPosInvalid THEN
			eInvertReqPos	:= eInvertCurrPos;
		END_IF
	ELSIF p_usiLinkProdRcpCurrRcpMcMod = 1 THEN //Inverter Mode
		IF bStepEntToInOff = TRUE AND p_bLinkConvHvBrd = TRUE THEN
			eInvertReqPos	:= InvertCurrPosAtHome;
		ELSIF bStepEntToEnd = TRUE AND p_bLinkConvHvBrd = TRUE THEN
			eInvertReqPos	:= InvertCurrPosAtRemote;
		END_IF

	ELSIF p_usiLinkProdRcpCurrRcpMcMod = 2 THEN // Invert Once Mode

		IF bInvOnceTwicePCBOut = FALSE THEN
			IF eInvertCurrPos <> InvertPosInvalid THEN
				eInvertReqPos	:= eInvertCurrPos;
			END_IF
		ELSE
			IF bStepInvRtrnEntToEnd = TRUE AND p_bLinkConvHvBrd = TRUE THEN
				eInvertReqPos	:= InvertCurrPosAtHome;
			ELSIF bStepInvRtrnEntToInOff = TRUE AND p_bLinkConvHvBrd = TRUE THEN
				eInvertReqPos	:= InvertCurrPosAtRemote;
			END_IF
		END_IF

	ELSIF p_usiLinkProdRcpCurrRcpMcMod = 3 THEN // Invert Twice Mode
		IF bStepEntToInOff = TRUE AND p_bLinkConvHvBrd = TRUE AND bInvOnceTwicePCBOut = FALSE THEN
			eInvertReqPos	:= InvertCurrPosAtHome;
		ELSIF bStepEntToEnd = TRUE AND p_bLinkConvHvBrd = TRUE AND bInvOnceTwicePCBOut = FALSE THEN
			eInvertReqPos	:= InvertCurrPosAtRemote;
		ELSIF bStepInvRtrnEntToEnd = TRUE AND p_bLinkConvHvBrd = TRUE AND bInvOnceTwicePCBOut = TRUE THEN
			eInvertReqPos	:=  InvertCurrPosAtHome;
		ELSIF bStepInvRtrnEntToInOff = TRUE AND p_bLinkConvHvBrd = TRUE AND bInvOnceTwicePCBOut = TRUE THEN
			eInvertReqPos	:=  InvertCurrPosAtRemote;
		END_IF
	ELSIF p_usiLinkProdRcpCurrRcpMcMod = 4 THEN
	//	bReversalTransport
		IF NOT(p_iHermesAction = 1) THEN
			IF eInvertCurrPos <> InvertPosInvalid THEN //as a bypass
				eInvertReqPos	:= eInvertCurrPos;
			END_IF
		ELSE //when action = 1
			IF bStepEntToInOff = TRUE  AND p_bUSReversal = FALSE AND EDGEPOS(p_bLinkConvHvBrd)  THEN
				eInvertReqPos	:= InvertCurrPosAtHome;
			ELSIF bStepEntToEnd = TRUE  AND p_bUSReversal = FALSE AND EDGEPOS(p_bLinkConvHvBrd) THEN
				eInvertReqPos	:= InvertCurrPosAtRemote;
			ELSIF bStepEntToEnd = TRUE AND p_bUSReversal = TRUE AND EDGEPOS(p_bLinkConvHvBrd)  THEN //enter from Rear US
				eInvertReqPos	:=  InvertCurrPosAtHome;
			ELSIF bStepEntToInOff = TRUE AND p_bUSReversal = TRUE AND EDGEPOS(p_bLinkConvHvBrd)  THEN
				eInvertReqPos	:=  InvertCurrPosAtRemote;
			END_IF
		END_IF
	END_IF

	IF p_bUSReversal THEN
		p_bUSHermesTransporting ACCESS p_USHermes2Transporting;
		p_bUSHermesStopTransport ACCESS p_USHermes2StopTransport;
	ELSE
		p_bUSHermesTransporting ACCESS p_USHermesTransporting;
		p_bUSHermesStopTransport ACCESS p_USHermesStopTransport;
	END_IF
	bReverseStoppingPos := p_bHermesEntToReversePosition; // XOR p_bUSReversal;

	//Update Current Invert Position
	IF p_bLinkInvertHomeSen = TRUE AND p_bLinkInvertRemoteSen = FALSE THEN
		eInvertCurrPos	:= InvertCurrPosAtHome;
	ELSIF p_bLinkInvertHomeSen = FALSE AND p_bLinkInvertRemoteSen = TRUE THEN
		eInvertCurrPos	:= InvertCurrPosAtRemote;
	ELSE
		eInvertCurrPos	:= InvertPosInvalid;
	END_IF

	//Update Invert Complete
	bInvertCompl	:= (eInvertCurrPos = eInvertReqPos) AND (eInvertReqPos <> InvertPosInvalid);

	//Update Pneumatic when change rcp prompt externally (leader follower change recipe)
	IF p_bRun THEN
		IF p_usiLinkProdRcpCurrRcpMcMod = 0 THEN
			bChangeInvertExtPneu	:= TRUE;
		ELSIF p_usiLinkProdRcpCurrRcpMcMod = 1 THEN
			bChangeBypassRetPneu	:= TRUE;
		END_IF
	END_IF

	IF bChangeBypassRetPneu AND p_usiLinkProdRcpCurrRcpMcMod = 0 AND eOpsStep>=InvertStepUSCommTmr THEN
		eStopperAct		:= PneuActRet;
		eOutletShutterAct:= PneuActRet;

		IF (p_eStopperStatus = Done AND p_eStopperStat = PneuActRet) AND (p_eOutletShutterStatus = Done AND p_eOutletShutterStat = PneuActRet)   THEN
			eStopperAct			:= PneuActIdle;
			eOutletShutterAct	:= PneuActIdle;
			bChangeBypassRetPneu:= FALSE;
		END_IF
	END_IF

	IF bChangeInvertExtPneu  AND  p_usiLinkProdRcpCurrRcpMcMod = 1  AND eOpsStep>=InvertStepUSCommTmr THEN

		IF eInvertCurrPos= InvertCurrPosAtHome THEN
			eStopperAct			:= PneuActExt;
			eOutletShutterAct	:= PneuActExt;

			IF (p_eStopperStatus = Done AND p_eStopperStat = PneuActExt) AND (p_eOutletShutterStatus = Done AND p_eOutletShutterStat = PneuActExt)   THEN
				eStopperAct			:= PneuActIdle;
				eOutletShutterAct	:= PneuActIdle;
				bChangeInvertExtPneu:= FALSE;
			END_IF
		ELSE
			bChangeInvertExtPneu:= FALSE;
		END_IF
	END_IF

	// Board In Memory from Upstream 1 for Invert One and Twice Mode
	IF (p_usiLinkProdRcpCurrRcpMcMod = 2 OR p_usiLinkProdRcpCurrRcpMcMod = 3) AND eOpsStep>InvertStepUSCommTmr AND bHvBrd AND bInvOnceTwicePCBOut = FALSE THEN
		bBoardInFromUS1	:= TRUE;
	ELSIF (p_usiLinkProdRcpCurrRcpMcMod = 2 OR p_usiLinkProdRcpCurrRcpMcMod = 3) AND bInvOnceTwicePCBOut THEN
		bBoardInFromUS1 := FALSE;
	END_IF

	//Reset Return Board from Reset Buttom
	IF p_bLinkUIRtnBrdReset  THEN
		bInvOnceTwicePCBOut := FALSE;
	END_IF

	//Waiting Return Board Status
	IF bInvOnceTwicePCBOut AND bStepInvRtrnUSCommTmr THEN
		udiStatus1 	:= 10009;
	ELSIF bInvOnceTwicePCBOut AND bStepDSCommTmr THEN
		udiStatus1	:= 10010;
	ELSIF bInvOnceTwicePCBOut THEN
		udiStatus1 	:= 10009;
	ELSE
		udiStatus1 	:= 0;
	END_IF

END_ACTION
```

#### Cyclic.st - Do Not Change!!!
```iecst
(** 2019-03-22 **)
PROGRAM _CYCLIC

	IF bInitDone = FALSE THEN
		bInitDone	:= TRUE;

		Act_InitLocal;
		Act_InitGlobal;

	ELSIF bInitialDone = FALSE THEN
		IF p_bNtSettingsLoadDone = TRUE THEN
			bInitialDone	:= TRUE;

			Act_Initial;
		END_IF

	ELSE

		Act_RstErr;
		Act_LinkEn;
		Act_Link;
		Act_Background;
		Act_Alarm;
		Act_AlarmInfo;

	END_IF

END_PROGRAM
```

#### Act_RstErr.st - Do Not Change!!!
```iecst
(** 2019-01-11 **)
ACTION Act_RstErr:

	IF p_udiRstErr <> udiRstErrOld THEN
		bRstErr			:= TRUE;
		udiRstErrOld	:= p_udiRstErr;
	ELSE
		bRstErr			:= FALSE;
	END_IF

END_ACTION
```

#### Act_InitLocal.st - Do Not Change!!!
```iecst
(** 2020-10-06 **)
ACTION Act_InitLocal:

	//Input Reference Link To Local Variable
	p_udiRstErr ACCESS ADR(udiRstErr);
	p_bEn ACCESS ADR(bEn);
	p_bDis ACCESS ADR(bDis);
	p_bRun ACCESS ADR(bRun);
	p_bStop ACCESS ADR(bStop);
	p_bStep ACCESS ADR(bStep);

	p_bInitGdBrd ACCESS ADR(bInitGdBrd);
	p_bInsertGdBrd ACCESS ADR(bInsertGdBrd);
	p_eConvDirection ACCESS ADR(eConvDirection);
	p_eUSCommMod ACCESS ADR(eUSCommMod);
	p_eDSCommMod ACCESS ADR(eDSCommMod);
	p_bGoToStandby ACCESS ADR(bGoToStandby);
	p_bUSAllow ACCESS ADR(bUSAllow);
	p_bDSAllow ACCESS ADR(bDSAllow);

	p_bRtrnUSAllow ACCESS ADR(bRtrnUSAllow);
	p_bRtrnDSAllow ACCESS ADR(bRtrnDSAllow);

	p_bLeftSen ACCESS ADR(bLeftSen);
	p_bRightSen ACCESS ADR(bRightSen);
	p_bMidSen ACCESS ADR(bMidSen);

	p_eUSSMEMAStat	ACCESS ADR(eUSSMEMAStat);
	p_eUSSMEMAStatus ACCESS ADR(eUSSMEMAStatus);
	p_bUSSMEMATransporting ACCESS ADR(bUSSMEMATransporting);
	p_bUSSMEMAConvStart ACCESS ADR(bUSSMEMAConvStart);
	p_bUSSMEMAConvStop ACCESS ADR(bUSSMEMAConvStop);
	p_bUSSMEMAUSRdy ACCESS ADR(bUSSMEMAUSRdy);
	p_bUSSMEMAUSGdBrdRdy ACCESS ADR(bUSSMEMAUSGdBrdRdy);

	p_eDSSMEMAStat	ACCESS ADR(eDSSMEMAStat);
	p_eDSSMEMAStatus ACCESS ADR(eDSSMEMAStatus);
	p_bDSSMEMAConvStart ACCESS ADR(bDSSMEMAConvStart);
	p_bDSSMEMAConvStop ACCESS ADR(bDSSMEMAConvStop);
	p_bDSSMEMATimer ACCESS ADR(bDSSMEMATimer);

	p_bUSHermesTransporting ACCESS ADR(bUSHermesTransporting);
	p_bUSHermesStopTransport ACCESS ADR(bUSHermesStopTransport);
	p_bUSHermesUSRdy ACCESS ADR(bUSHermesUSRdy);
	p_bUSHermesUSGdRdy ACCESS ADR(bUSHermesUSGdRdy);

	p_bDSHermesTransporting ACCESS ADR(bDSHermesTransporting);
	p_bDSHermesStopTransport ACCESS ADR(bDSHermesStopTransport);

	p_eConvStat	ACCESS ADR(eConvStat);
	p_eConvStatus ACCESS ADR(eConvStatus);
	p_bConvHvBrd ACCESS ADR(bConvHvBrd);

	p_eStopperStat ACCESS ADR(eStopperStat);
	p_eStopperStatus ACCESS ADR(eStopperStatus);
	p_bStopperExtended ACCESS ADR(bStopperExtended);
	p_bStopperRetracted ACCESS ADR(bStopperRetracted);

	p_eClampStat ACCESS ADR(eClampStat);
	p_eClampStatus ACCESS ADR(eClampStatus);

	p_eInletShutterStat ACCESS ADR(eInletShutterStat);
	p_eInletShutterStatus ACCESS ADR(eInletShutterStatus);
	p_bInletShutterOpen ACCESS ADR(bInletShutterOpen);
	p_bInletShutterClose ACCESS ADR(bInletShutterClose);

	p_eOutletShutterStat ACCESS ADR(eOutletShutterStat);
	p_eOutletShutterStatus ACCESS ADR(eOutletShutterStatus);
	p_bOutletShutterOpen ACCESS ADR(bOutletShutterOpen);
	p_bOutletShutterClose ACCESS ADR(bOutletShutterClose);

	p_eClamp1Stat ACCESS ADR (eClamp1Stat);
	p_eClamp1Status ACCESS ADR (eClamp1Status);
	p_bClampRS1 ACCESS ADR (bClampRS1);
	p_bUnClampRS1 ACCESS ADR ( bUnClampRS1);

	p_eClamp2Stat ACCESS ADR (eClamp2Stat);
	p_eClamp2Status ACCESS ADR (eClamp2Status);
	p_bClampRS2 ACCESS ADR (bClampRS2);
	p_bUnClampRS2 ACCESS ADR ( bUnClampRS2);

	p_eClamp3Stat ACCESS ADR (eClamp3Stat);
	p_eClamp3Status ACCESS ADR (eClamp3Status);
	p_bClampRS3 ACCESS ADR (bClampRS3);
	p_bUnClampRS3 ACCESS ADR ( bUnClampRS3);

	p_sProgNm ACCESS ADR(sProgNm);
	p_bNtSettingsLoadDone ACCESS ADR(bNtSettingsLoadDone);

	p_bClampDis ACCESS ADR(bClampDis);
	p_bClampPrep ACCESS ADR(bClampPrep);
	p_eClampOption ACCESS ADR(eClampOption);

	p_bInletShutterPrep ACCESS ADR(bInletShutterPrep);
	p_bInletShutterDis ACCESS ADR(bInletShutterDis);
	p_bOutletShutterPrep ACCESS ADR(bOutletShutterPrep);
	p_bOutletShutterDis ACCESS ADR(bOutletShutterDis);

	p_bClamp2Sen ACCESS ADR(bClamp2Sen);
	p_bClamp3Sen ACCESS ADR(bClamp3Sen);

	p_diFwdDlyTm ACCESS ADR(diFwdDlyTm);
	p_diRevDlyTm ACCESS ADR(diRevDlyTm);

END_ACTION
```

#### Act_Background.st - Do Not Change!!!
```iecst
(** 2019-04-16 **)
ACTION Act_Background:

	//Reset bPaused
	IF EDGENEG(p_bStop OR p_bStep) THEN
		bPaused	:= FALSE;
	END_IF

	IF eStatus <> Error AND p_bRun = TRUE THEN
		IF (p_bEn = TRUE) AND (p_bDis = FALSE) THEN
			Act_OpsRun;
		ELSE
			bPaused	:= p_bStop OR p_bStep;
		END_IF

		IF EDGEPOS(p_bEn = FALSE OR p_bDis = TRUE) THEN
			Act_OpsRst;
		END_IF

	ELSIF eStatus <> Error THEN
		sStepTxt	:= 'Stop';
	ELSE
		sStepTxt	:= 'Error';
	END_IF

	//Reset
	IF EDGENEG(p_bRun) OR EDGEPOS(eStatus = Error) THEN
		Act_OpsInitial;
		Act_OpsRst;
	END_IF

	//Reset Error
	IF (eStatus = Error) AND bRstErr THEN
		eStatus		:= Idle;
		udiStatus	:= 0;
	END_IF

END_ACTION
```

#### Act_Alarm.st - Do Not Change!!!
```iecst
(** 2019-03-25 **)
ACTION Act_Alarm:

	//Error
	IF EDGEPOS(eStatus = Error) THEN

		tyAlmData.sProgNm		:= p_sProgNm;
		tyAlmData.udiCode		:= udiStatus;
		tyAlmData.eSeverity		:= AlmSeverityError;
		tyAlmData.udiRunTime	:= tyAlmData.udiRunTime + 1;
		tyAlmData.bAlm			:= TRUE;
		tyAlmData.udiModuleNum  := udiModuleNum;
		g_sOpsInvertProgNm		:= p_sProgNm;

		//Get Error Message
		IF tyAlmData.udiCode < 10000 OR tyAlmData.udiCode > 10099 THEN
			tyAlmData.sAlmMsg	:= 'Unknown';
			tyAlmData.sRcyMsg	:= 'Unknown';
		ELSE
			tyAlmData.sAlmMsg	:= a_tyAlmText[tyAlmData.udiCode].sAlmText;
			tyAlmData.sRcyMsg	:= a_tyAlmText[tyAlmData.udiCode].sRcyText;
		END_IF

	ELSIF bRstErr AND (tyAlmData.udiCode <> 0) THEN

		tyAlmData.udiCode		:= 0;
		tyAlmData.eSeverity		:= AlmSeverityNA;
		tyAlmData.sAlmMsg		:= '';
		tyAlmData.sRcyMsg		:= '';
		tyAlmData.bAlm			:= FALSE;
	END_IF

END_ACTION
```

#### Act_AlarmInfo.st - Do Not Change!!!
```iecst
(** 2019-03-25 **)
ACTION Act_AlarmInfo:

	//Info
	tyAlmData1.sProgNm		:= p_sProgNm;
	tyAlmData1.udiCode		:= udiStatus1;
	tyAlmData1.eSeverity	:= AlmSeverityInfo;
	tyAlmData1.udiRunTime	:= tyAlmData1.udiRunTime + 1;
	tyAlmData.bAlm			:= TRUE;
	tyAlmData.udiModuleNum  := udiModuleNum;
	g_sOpsInvertProgNm		:= p_sProgNm;

	//Get Info Message
	IF tyAlmData1.udiCode < 10000 OR tyAlmData1.udiCode > 10099 THEN
		tyAlmData1.sAlmMsg	:= 'Unknown';
		tyAlmData1.sRcyMsg	:= 'Unknown';
	ELSE
		tyAlmData1.sAlmMsg	:= a_tyAlmText[tyAlmData1.udiCode].sAlmText;
		tyAlmData1.sRcyMsg	:= a_tyAlmText[tyAlmData1.udiCode].sRcyText;
	END_IF

END_ACTION
```

#### Package Logical/Operations/OpsInvert/Sequence - Change By Project

#### Act_OpsInitial.st - Do Not Change!!!
```iecst
(** 2019-01-16 **)
ACTION Act_OpsInitial:

	eOpsStep			:= InvertStepNA;
	eGotoOpsStep		:= InvertStepInitChkCondition;

	bStepInitConv		:= FALSE;
	bStepInitDone		:= FALSE;
	bStepUSStandby		:= FALSE;
	bStepUSCommTmr		:= FALSE;
	bStepEntToEnd		:= FALSE;
	bStepEntToInOff		:= FALSE;
	bStepRev			:= FALSE;
	bStepPreExit		:= FALSE;
	bStepDSStandby		:= FALSE;
	bStepDSCommTmr		:= FALSE;
	bStepExitBrd		:= FALSE;
	bStepSafeMode		:= FALSE;
	bStepInvRtrnEntToEnd	:= FALSE;
	bStepInvRtrnEntToInOff	:= FALSE;
	bStepInvRtrnUSStandby	:= FALSE;
	bStepInvRtrnUSCommTmr	:= FALSE;
END_ACTION
```

#### Act_OpsRun.st
```iecst
(** 2020-10-06 **)
ACTION Act_OpsRun:
	IF p_usiLinkProdRcpCurrRcpMcMod = 4 THEN
		Act_OpsStandard_Hermes;
	ELSIF (p_bClampPrep = FALSE) OR ((p_bClampPrep=TRUE) AND (p_eClampOption=ClampNoRS)) THEN

		Act_OpsStandard;

	ELSIF (p_usiLinkProdRcpCurrRcpMcMod = 2 OR p_usiLinkProdRcpCurrRcpMcMod = 3) THEN

		Act_OpsClampNoStopperInvOnceAndTwice;

	ELSE

		Act_OpsClampNoStopper;

	END_IF

END_ACTION
```

#### Act_OpsRst.st - Do Not Change!!!
```iecst
(** 2020-10-06 **)
ACTION Act_OpsRst:

	eUSSMEMAAct			:= SMEMAActIdle;
	eDSSMEMAAct			:= SMEMAActIdle;
	eConvAct			:= ConvActIdle;
	eStopperAct			:= PneuActIdle;
	eAWAct				:= AWActIdle;
	eClampAct			:= PneuActIdle;
	eInletShutterAct	:= PneuActIdle;
	eOutletShutterAct	:= PneuActIdle;
	eClamp1Act			:= PneuActIdle;
	eClamp2Act			:= PneuActIdle;
	eClamp3Act			:= PneuActIdle;
	eInvertAct			:= MotorBrkActIdle;
	eUSSMEMA2Act		:= SMEMAActIdle;

	bBrdInserted		:= FALSE;
	bBrdRemoved			:= FALSE;

	bUSTimerRun			:= FALSE;
	bDSTimerRun			:= FALSE;
	bReachedEnd			:= FALSE;
	bHvBrd				:= FALSE;
	bGdBrd				:= FALSE;
	bUS2TimerRun		:= FALSE;

	bClampDisInitUnblk	:= FALSE;
	bInvertPosInvalidSkipInit := FALSE;
	bChangeBypassRetPneu:= FALSE;
	bChangeInvertExtPneu:= FALSE;

	fbFwdTimer(IN := FALSE);
	fbRevTimer(IN := FALSE);

END_ACTION
```

#### Act_LogStep.st
```iecst
(** 2019-03-25 **)
ACTION Act_LogStep:

//log
	IF EDGEPOS (bClsLog) THEN
		memset(ADR(logStep),0,SIZEOF(logStep));
		logIndexStep := 0;
	END_IF

	blog := eOpsStep <> eGotoOpsStepDummy;

	IF blog THEN
		logStep[logIndexStep] := eOpsStep;
		logIndexStep := logIndexStep + 1;
		IF logIndexStep > SIZEOF(logStep)/SIZEOF(logStep[0]) -1 THEN
			logIndexStep := 0;
		END_IF
	END_IF

	eGotoOpsStepDummy := eOpsStep;

END_ACTION
```

#### Act_OpsStandard.st
```iecst
(** 2020-10-06 **)
ACTION Act_OpsStandard:

	IF eGotoOpsStep <> eOpsStep THEN

		CASE eGotoOpsStep OF

			ELSE
				eOpsStep	:= eGotoOpsStep;

		END_CASE

	END_IF

	IF eOpsStep = eGotoOpsStep THEN

		IF bPaused = FALSE THEN

			CASE eOpsStep OF

				InvertStepInitChkCondition:
					sStepTxt	:= 'Init Check Condition';

					IF p_bClampPrep THEN
						IF eInvertCurrPos	= InvertPosInvalid THEN
							bInvertPosInvalidSkipInit := TRUE;

							IF p_bClampDis THEN
								bClampDisInitUnblk	:= TRUE;
							END_IF

							eGotoOpsStep	:= InvertStepClampBlkBefInvert;
						ELSE
							eGotoOpsStep	:= InvertStepInitClampUnblk;
						END_IF
					ELSE
						IF eInvertCurrPos	= InvertPosInvalid THEN
							bInvertPosInvalidSkipInit := TRUE;

							IF (p_bInletShutterPrep AND p_bInletShutterDis=FALSE) OR (p_bOutletShutterPrep AND p_bOutletShutterDis=FALSE) THEN
								eGotoOpsStep	:= InvertStepShuttersCloseBefInvert;
							ELSE
								eGotoOpsStep	:= InvertStepInvert;
							END_IF
						ELSE
							eGotoOpsStep	:= InvertStepInitInvertComplChk;
						END_IF
					END_IF

					bPaused	:= p_bStop OR p_bStep;

				InvertStepInitClampUnblk:
					sStepTxt	:= 'Init Clamp Unblock';

					eClampAct	:= PneuActRet;

					IF p_eClampStatus = Done AND p_eClampStat = PneuActRet THEN

						eClampAct		:= PneuActIdle;
						eGotoOpsStep	:= InvertStepInitInvertComplChk;

						bPaused	:= p_bStop OR p_bStep;
					END_IF

				InvertStepInitInvertComplChk:
					sStepTxt	:= 'Init Checking Invert Complete Condition';

					IF bInvertCompl = FALSE THEN
						IF eInvertCurrPos = InvertCurrPosAtRemote THEN
							IF p_bLeftSen = TRUE THEN
								eGotoOpsStep	:= InvertStepInitConvAwayLftSen;
							ELSE
								eGotoOpsStep	:= InvertStepInitStopperBlk;
							END_IF

						ELSIF eInvertCurrPos = InvertCurrPosAtHome THEN
							IF p_bRightSen = TRUE THEN
								eGotoOpsStep	:= InvertStepInitConvAwayRgtSen;
							ELSE
								eGotoOpsStep	:= InvertStepInitStopperBlk;
							END_IF

						ELSE
							eGotoOpsStep	:= InvertStepInitStopperBlk;
						END_IF

					ELSE
						eGotoOpsStep	:= InvertStepInitStopperUnblk;
					END_IF

					bPaused	:= p_bStop OR p_bStep;

				InvertStepInitConvAwayLftSen:
					sStepTxt	:= 'Init Conveyor Away Stopper At Left';

					eConvAct	:= ConvActInit;

					fbFwdTimer(IN := TRUE, PT := DINT_TO_TIME(p_diFwdDlyTm));

					IF fbFwdTimer.Q = TRUE THEN
						fbFwdTimer(IN := FALSE);

						bHvBrd			:= FALSE;
						p_bConvHvBrd	:= FALSE;

						eConvAct		:= ConvActIdle;

						eGotoOpsStep	:= InvertStepInitStopperBlk;

						bPaused	:= p_bStop OR p_bStep;

					ELSIF p_eConvStatus = Done AND p_eConvStat = ConvActInit THEN
						fbFwdTimer(IN := FALSE);

						bHvBrd 			:= TRUE;
						bGdBrd			:= p_bInitGdBrd;

						eConvAct		:= ConvActIdle;

						eGotoOpsStep	:= InvertStepInitStopperBlk;

						bPaused	:= p_bStop OR p_bStep;
					END_IF

				InvertStepInitConvAwayRgtSen:
					sStepTxt	:= 'Init Conveyor Away Stopper At Right';

					eConvAct	:= ConvActRevImmedStart;

					fbRevTimer(IN := TRUE, PT := DINT_TO_TIME(p_diRevDlyTm));

					IF fbRevTimer.Q = TRUE THEN
						fbRevTimer(IN := FALSE);

						bHvBrd			:= FALSE;
						p_bConvHvBrd	:= FALSE;

						eConvAct		:= ConvActIdle;

						eGotoOpsStep	:= InvertStepInitStopperBlk;

						bPaused	:= p_bStop OR p_bStep;

					ELSIF p_eConvStatus = Done AND p_eConvStat = ConvActRevImmedStart THEN
						fbRevTimer(IN := FALSE);

						bHvBrd 			:= TRUE;
						bGdBrd			:= p_bInitGdBrd;

						eConvAct		:= ConvActIdle;

						eGotoOpsStep	:= InvertStepInitStopperBlk;

						bPaused	:= p_bStop OR p_bStep;
					END_IF

				InvertStepInitStopperBlk:
					sStepTxt	:= 'Init Stopper Block';

					eStopperAct	:= PneuActExt;

					IF p_eStopperStatus = Done AND p_eStopperStat = PneuActExt THEN
						eStopperAct := PneuActIdle;

						IF eInvertCurrPos = InvertCurrPosAtRemote THEN
							eGotoOpsStep  := InvertStepInitConvTwdLftSen;

						ELSIF eInvertCurrPos = InvertCurrPosAtHome THEN
							eGotoOpsStep  := InvertStepInitConvTwdRgtSen;
						END_IF

						bPaused	:= p_bStop OR p_bStep;
					END_IF

				InvertStepInitConvTwdLftSen:
					sStepTxt	:= 'Init Conveyor Toward Stopper At Left';

					eConvAct	:= ConvActRevImmedStart;

					fbRevTimer(IN := TRUE, PT := DINT_TO_TIME(p_diRevDlyTm));

					IF fbRevTimer.Q = TRUE THEN
						fbRevTimer(IN := FALSE);

						bHvBrd			:= FALSE;
						p_bConvHvBrd	:= FALSE;

						eConvAct		:= ConvActIdle;

						IF p_bClampPrep AND p_bClampDis=FALSE THEN
							eGotoOpsStep	:= InvertStepClampBlkBefInvert;
						ELSE
							IF (p_bInletShutterPrep AND p_bInletShutterDis=FALSE) OR (p_bOutletShutterPrep AND p_bOutletShutterDis=FALSE) THEN
								eGotoOpsStep	:= InvertStepShuttersCloseBefInvert;
							ELSE
								eGotoOpsStep	:= InvertStepInvert;
							END_IF
						END_IF

						bPaused	:= p_bStop OR p_bStep;

					ELSIF p_eConvStatus = Done AND p_eConvStat = ConvActRevImmedStart THEN
						fbRevTimer(IN := FALSE);
						eConvAct	:= ConvActIdle;

						bHvBrd			:= TRUE;
						bGdBrd			:= p_bInitGdBrd;

						IF p_bClampPrep AND p_bClampDis=FALSE THEN
							eGotoOpsStep	:= InvertStepClampBlkBefInvert;
						ELSE
							IF (p_bInletShutterPrep AND p_bInletShutterDis=FALSE) OR (p_bOutletShutterPrep AND p_bOutletShutterDis=FALSE) THEN
								eGotoOpsStep	:= InvertStepShuttersCloseBefInvert;
							ELSE
								eGotoOpsStep	:= InvertStepInvert;
							END_IF
						END_IF

						bPaused	:= p_bStop OR p_bStep;

					END_IF

				InvertStepInitConvTwdRgtSen:
					sStepTxt	:= 'Init Conveyor Toward Stopper at Right';

					eConvAct	:= ConvActInit;

					fbFwdTimer(IN := TRUE, PT := DINT_TO_TIME(p_diFwdDlyTm));

					IF fbFwdTimer.Q = TRUE THEN
						fbFwdTimer(IN := FALSE);

						bHvBrd			:= FALSE;
						p_bConvHvBrd	:= FALSE;

						eConvAct	:= ConvActIdle;

						IF p_bClampPrep AND p_bClampDis=FALSE THEN
							eGotoOpsStep	:= InvertStepClampBlkBefInvert;
						ELSE
							IF (p_bInletShutterPrep AND p_bInletShutterDis=FALSE) OR (p_bOutletShutterPrep AND p_bOutletShutterDis=FALSE) THEN
								eGotoOpsStep	:= InvertStepShuttersCloseBefInvert;
							ELSE
								eGotoOpsStep	:= InvertStepInvert;
							END_IF
						END_IF

						bPaused	:= p_bStop OR p_bStep;

					ELSIF p_eConvStatus = Done AND p_eConvStat = ConvActInit THEN
						fbFwdTimer(IN := FALSE);
						eConvAct	:= ConvActIdle;

						bHvBrd			:= TRUE;
						bGdBrd			:= p_bInitGdBrd;

						IF p_bClampPrep AND p_bClampDis=FALSE THEN
							eGotoOpsStep	:= InvertStepClampBlkBefInvert;
						ELSE
							IF (p_bInletShutterPrep AND p_bInletShutterDis=FALSE) OR (p_bOutletShutterPrep AND p_bOutletShutterDis=FALSE) THEN
								eGotoOpsStep	:= InvertStepShuttersCloseBefInvert;
							ELSE
								eGotoOpsStep	:= InvertStepInvert;
							END_IF
						END_IF

						bPaused	:= p_bStop OR p_bStep;
					END_IF

				InvertStepInitStopperUnblk:
					sStepTxt	:= 'Init Stopper Unblock';

					eStopperAct	:= PneuActRet;

					IF p_eStopperStatus = Done AND p_eStopperStat = PneuActRet THEN
						eStopperAct		:= PneuActIdle;
						eGotoOpsStep	:= InvertStepInitConvToRgt;

						bPaused	:= p_bStop OR p_bStep;
					END_IF

				InvertStepInitConvToRgt:
					sStepTxt	:= 'Init Conveyor to Right';

					eConvAct	:= ConvActInit;

					IF p_eConvStatus = Done AND p_eConvStat = ConvActInit THEN
						eConvAct		:= ConvActIdle;

						IF (p_bInletShutterPrep AND p_bInletShutterDis=FALSE) OR (p_bOutletShutterPrep AND p_bOutletShutterDis=FALSE) THEN
							eGotoOpsStep	:= InvertStepInitShuttersInOutClose;
						ELSE
							IF p_bRightSen = TRUE THEN

								bHvBrd 	:= TRUE;
								bGdBrd	:= p_bInitGdBrd;

								eGotoOpsStep	:= InvertStepDSStandby;
							ELSE
								IF p_bAWWidthPosDiff = TRUE THEN
									eGotoOpsStep	:= InvertStepAWMov;
								ELSE
									eGotoOpsStep	:= InvertStepChkCondition;
								END_IF
							END_IF

						END_IF

						bPaused	:= p_bStop OR p_bStep;
					END_IF

				InvertStepInitShuttersInOutClose:
					sStepTxt			:= 'Init Closing Shutters';

					eInletShutterAct	:= PneuActExt;
					eOutletShutterAct	:= PneuActExt;

					IF (p_eInletShutterStatus = Done AND p_eInletShutterStat = PneuActExt) AND (p_eOutletShutterStatus = Done AND p_eOutletShutterStat = PneuActExt) THEN

						eInletShutterAct	:= PneuActIdle;
						eOutletShutterAct	:= PneuActIdle;

						IF p_bRightSen = TRUE THEN

							bHvBrd 	:= TRUE;
							bGdBrd	:= p_bInitGdBrd;

							IF p_bOutletShutterOpen THEN
								eGotoOpsStep	:= InvertStepDSStandby;
							ELSE
								IF p_usiLinkProdRcpCurrRcpMcMod=0 THEN
									eGotoOpsStep	:= InvertStepDSInOutletShutterOpen;
								ELSE
									eGotoOpsStep	:= InvertStepOutletShutterOpen;
								END_IF
							END_IF

						ELSE
							IF p_bAWWidthPosDiff = TRUE THEN
								eGotoOpsStep	:= InvertStepAWMov;
							ELSE
								eGotoOpsStep	:= InvertStepChkCondition;
							END_IF
						END_IF

						bPaused	:= p_bStop OR p_bStep;
					END_IF

				InvertStepShuttersInOutClose:
					sStepTxt			:= 'Closing Shutters Prior to Auto Width Change';

					eInletShutterAct	:= PneuActExt;
					eOutletShutterAct	:= PneuActExt;

					IF (p_eInletShutterStatus = Done AND p_eInletShutterStat = PneuActExt) AND (p_eOutletShutterStatus = Done AND p_eOutletShutterStat = PneuActExt) THEN

						eInletShutterAct	:= PneuActIdle;
						eOutletShutterAct	:= PneuActIdle;

						eGotoOpsStep	:= InvertStepAWMov;

						bPaused	:= p_bStop OR p_bStep;
					END_IF

				InvertStepAWMov:
					sStepTxt	:= 'Moving Auto Width';

					eAWAct	:= AWActGoWidthOff;

					IF p_eAWStatus = Done AND p_eAWStat = AWActGoWidthOff THEN
						eAWAct			:= AWActIdle;

						eGotoOpsStep	:= InvertStepChkCondition;

						bPaused	:= p_bStop OR p_bStep;
					END_IF

				InvertStepChkCondition:
					sStepTxt	:= 'Check Condition';

					IF (p_bInletShutterPrep AND p_bInletShutterDis=FALSE) OR (p_bOutletShutterPrep AND p_bOutletShutterDis=FALSE) THEN
						IF p_bUSAllow THEN
							eGotoOpsStep	:= InvertStepChkShutterCond;
						END_IF
					ELSE
						eGotoOpsStep	:= InvertStepStopperPosChk;
					END_IF

					bPaused	:= p_bStop OR p_bStep;

				InvertStepChkShutterCond:
					sStepTxt	:= 'Check Initial Shutter Condition';

					IF p_usiLinkProdRcpCurrRcpMcMod = 0 THEN
						IF p_bInletShutterOpen AND p_bOutletShutterOpen THEN
							eGotoOpsStep:= InvertStepStopperPosChk;
						ELSE
							eGotoOpsStep:= InvertStepShuttersInOutOpen;
						END_IF
					ELSIF p_usiLinkProdRcpCurrRcpMcMod = 1 THEN
						IF p_bInletShutterOpen AND p_bOutletShutterClose THEN
							eGotoOpsStep:= InvertStepStopperPosChk;
						ELSE
							eGotoOpsStep:= InvertStepShuttersInOpenOutClose;
						END_IF

					END_IF

					bPaused	:= p_bStop OR p_bStep;

					//Open both shutters if bypass mode
				InvertStepShuttersInOutOpen:
					sStepTxt			:= 'Opening Shutters Prior After Auto Width Change';

					eInletShutterAct	:= PneuActRet;
					eOutletShutterAct	:= PneuActRet;

					IF (p_eInletShutterStatus = Done AND p_eInletShutterStat = PneuActRet) AND (p_eOutletShutterStatus = Done AND p_eOutletShutterStat = PneuActRet) THEN

						eInletShutterAct	:= PneuActIdle;
						eOutletShutterAct	:= PneuActIdle;

						eGotoOpsStep	:= InvertStepStopperPosChk;

						bPaused	:= p_bStop OR p_bStep;
					END_IF

					//Open inlet shutter close outlet if invert mode
				InvertStepShuttersInOpenOutClose:
					sStepTxt			:= 'Opening Inlet Shutter and Closing Outlet Shutter';

					eInletShutterAct	:= PneuActRet;
					eOutletShutterAct	:= PneuActExt;

					IF (p_eInletShutterStatus = Done AND p_eInletShutterStat = PneuActRet) AND (p_eOutletShutterStatus = Done AND p_eOutletShutterStat = PneuActExt) THEN

						eInletShutterAct	:= PneuActIdle;
						eOutletShutterAct	:= PneuActIdle;

						eGotoOpsStep	:= InvertStepStopperPosChk;

						bPaused	:= p_bStop OR p_bStep;
					END_IF

				InvertStepStopperPosChk:
					sStepTxt	:= 'Checking Stopper Position';

					IF eInvertCurrPos = InvertCurrPosAtRemote THEN
						eGotoOpsStep	:= InvertStepStopperUnblk;

					ELSIF eInvertCurrPos = InvertCurrPosAtHome THEN
						IF p_usiLinkProdRcpCurrRcpMcMod = 0 THEN
							eGotoOpsStep	:= InvertStepStopperUnblk;
						ELSIF p_usiLinkProdRcpCurrRcpMcMod = 1 THEN
							eGotoOpsStep	:= InvertStepStopperBlk;
						END_IF

					END_IF

					bPaused	:= p_bStop OR p_bStep;

				InvertStepStopperBlk:
					sStepTxt	:= 'Stopper Block';

					eStopperAct	:= PneuActExt;

					IF p_eStopperStatus = Done AND p_eStopperStat = PneuActExt THEN
						eStopperAct		:= PneuActIdle;
						eGotoOpsStep	:= InvertStepUSStandby;

						bPaused	:= p_bStop OR p_bStep;
					END_IF

				InvertStepStopperUnblk:
					sStepTxt	:= 'Stopper Unblock';

					eStopperAct	:= PneuActRet;

					IF p_eStopperStatus = Done AND p_eStopperStat = PneuActRet THEN
						eStopperAct		:= PneuActIdle;
						eGotoOpsStep	:= InvertStepUSStandby;

						bPaused	:= p_bStop OR p_bStep;
					END_IF

				InvertStepUSStandby:
					sStepTxt	:= 'In Upstream Standby Condition';

					bUSTimerRun	:= FALSE;

					bConvSen	:= p_bLeftSen OR p_bRightSen OR p_bMidSen;

					IF p_bAWWidthPosDiff = TRUE THEN
						IF (p_bInletShutterPrep AND p_bInletShutterDis=FALSE) OR (p_bOutletShutterPrep AND p_bOutletShutterDis=FALSE) THEN
							eGotoOpsStep	:= InvertStepShuttersInOutClose;
						ELSE
							eGotoOpsStep	:= InvertStepAWMov;
						END_IF
					ELSIF p_bUSAllow = TRUE THEN
						eGotoOpsStep	:= InvertStepUSCommTmr;
					ELSIF bConvSen = TRUE THEN
						eGotoOpsStep	:= InvertStepUSTmr;
					END_IF

					bPaused	:= p_bStop OR p_bStep;

				InvertStepUSTmr:
					sStepTxt	:= 'Inserting Board By Timer';

					bConvSen	:= p_bLeftSen OR p_bRightSen OR p_bMidSen;

					fbUSTimer(IN := bConvSen);

					IF fbUSTimer.Q = TRUE THEN
						bUSTimerRun	:= TRUE;
						fbUSTimer(IN := FALSE);

						bGdBrd	:= p_bInsertGdBrd;

						IF p_usiLinkProdRcpCurrRcpMcMod = 0 THEN
							eGotoOpsStep	:= InvertStepEntToEnd;

						ELSIF p_usiLinkProdRcpCurrRcpMcMod = 1 THEN
							IF eInvertCurrPos = InvertCurrPosAtRemote THEN
								eGotoOpsStep	:= InvertStepEntToInOff;
							ELSIF eInvertCurrPos = InvertCurrPosAtHome THEN
								eGotoOpsStep	:= InvertStepEntToEnd;
							END_IF

						END_IF

					ELSIF bConvSen = FALSE THEN
						bUSTimerRun	:= FALSE;
						fbUSTimer(IN := FALSE);

						IF p_bAWWidthPosDiff = TRUE THEN
							IF (p_bInletShutterPrep AND p_bInletShutterDis=FALSE) OR (p_bOutletShutterPrep AND p_bOutletShutterDis=FALSE) THEN
								eGotoOpsStep	:= InvertStepShuttersInOutClose;
							ELSE
								eGotoOpsStep	:= InvertStepAWMov;
							END_IF
						ELSE
							eGotoOpsStep	:= InvertStepUSStandby;
						END_IF

					ELSE
						bPaused	:= p_bStop;

						IF bPaused = TRUE THEN
							bUSTimerRun	:= FALSE;
							fbUSTimer(IN := FALSE);

							eGotoOpsStep	:= InvertStepUSStandby;
						END_IF

					END_IF

				InvertStepUSCommTmr:
					sStepTxt	:= 'Communicating Upstream Machine';

					CASE p_eUSCommMod OF
						McSetCommModSMEMA:
							fbUSTimer(IN := p_bLeftSen OR p_bRightSen OR p_bMidSen);

							eUSSMEMAAct	:= SMEMAActRun;

							IF p_bUSSMEMATransporting = TRUE THEN
								bUSTimerRun	:= FALSE;
								fbUSTimer(IN := FALSE);

								bGdBrd			:= p_bUSSMEMAUSGdBrdRdy;

								sStepTxt		:= 'Conveyor Entering Board';

								IF p_usiLinkProdRcpCurrRcpMcMod = 0 THEN
									eGotoOpsStep	:= InvertStepEntToEnd;

								ELSIF p_usiLinkProdRcpCurrRcpMcMod = 1 THEN
									IF eInvertCurrPos = InvertCurrPosAtRemote THEN
										eGotoOpsStep	:= InvertStepEntToInOff;
									ELSIF eInvertCurrPos = InvertCurrPosAtHome THEN
										eGotoOpsStep	:= InvertStepEntToEnd;
									END_IF

								END_IF

							ELSIF fbUSTimer.Q = TRUE THEN
								bUSTimerRun	:= TRUE;
								fbUSTimer(IN := FALSE);

								bGdBrd	:= p_bInsertGdBrd;

								IF p_usiLinkProdRcpCurrRcpMcMod = 0 THEN
									eGotoOpsStep	:= InvertStepEntToEnd;

								ELSIF p_usiLinkProdRcpCurrRcpMcMod = 1 THEN
									IF eInvertCurrPos = InvertCurrPosAtRemote THEN
										eGotoOpsStep	:= InvertStepEntToInOff;
									ELSIF eInvertCurrPos = InvertCurrPosAtHome THEN
										eGotoOpsStep	:= InvertStepEntToEnd;
									END_IF

								END_IF

							ELSIF (p_bAWWidthPosDiff = TRUE) OR (p_bUSAllow = FALSE) THEN
								bUSTimerRun	:= FALSE;
								fbUSTimer(IN := FALSE);

								eUSSMEMAAct	:= SMEMAActIdle;

								IF p_bAWWidthPosDiff = TRUE THEN
									IF (p_bInletShutterPrep AND p_bInletShutterDis=FALSE) OR (p_bOutletShutterPrep AND p_bOutletShutterDis=FALSE) THEN
										eGotoOpsStep	:= InvertStepShuttersInOutClose;
									ELSE
										eGotoOpsStep	:= InvertStepAWMov;
									END_IF
								ELSE
									eGotoOpsStep	:= InvertStepUSStandby;
								END_IF

							ELSE

								bPaused	:= p_bStop;

								IF bPaused = TRUE THEN
									bUSTimerRun	:= FALSE;
									fbUSTimer(IN := FALSE);

									eUSSMEMAAct	:= SMEMAActIdle;

									eGotoOpsStep	:= InvertStepUSStandby;
								END_IF

							END_IF

						McSetCommModHermes:
							fbUSTimer(IN := p_bLeftSen OR p_bRightSen OR p_bMidSen);

							IF p_bUSHermesTransporting = TRUE THEN
								bUSTimerRun	:= FALSE;
								fbUSTimer(IN := FALSE);

								bGdBrd	:= p_bUSHermesUSGdRdy;

								IF p_usiLinkProdRcpCurrRcpMcMod = 0 THEN
									eGotoOpsStep	:= InvertStepEntToEnd;

								ELSIF p_usiLinkProdRcpCurrRcpMcMod = 1 THEN
									IF eInvertCurrPos = InvertCurrPosAtRemote THEN
										eGotoOpsStep	:= InvertStepEntToInOff;
									ELSIF eInvertCurrPos = InvertCurrPosAtHome THEN
										eGotoOpsStep	:= InvertStepEntToEnd;
									END_IF

								END_IF

							ELSIF fbUSTimer.Q = TRUE THEN
								bUSTimerRun	:= TRUE;
								fbUSTimer(IN := FALSE);

								bGdBrd	:= p_bInsertGdBrd;

								IF p_usiLinkProdRcpCurrRcpMcMod = 0 THEN
									eGotoOpsStep	:= InvertStepEntToEnd;

								ELSIF p_usiLinkProdRcpCurrRcpMcMod = 1 THEN
									IF eInvertCurrPos = InvertCurrPosAtRemote THEN
										eGotoOpsStep	:= InvertStepEntToInOff;
									ELSIF eInvertCurrPos = InvertCurrPosAtHome THEN
										eGotoOpsStep	:= InvertStepEntToEnd;
									END_IF

								END_IF

							ELSIF (p_bAWWidthPosDiff = TRUE) OR (p_bUSAllow = FALSE) THEN
								bUSTimerRun	:= FALSE;
								fbUSTimer(IN := FALSE);

								IF p_bAWWidthPosDiff = TRUE THEN
									IF (p_bInletShutterPrep AND p_bInletShutterDis=FALSE) OR (p_bOutletShutterPrep AND p_bOutletShutterDis=FALSE) THEN
										eGotoOpsStep	:= InvertStepShuttersInOutClose;
									ELSE
										eGotoOpsStep	:= InvertStepAWMov;
									END_IF
								ELSE
									eGotoOpsStep	:= InvertStepUSStandby;
								END_IF

							ELSE

								bPaused	:= p_bStop;

								IF bPaused = TRUE THEN
									bUSTimerRun	:= FALSE;
									fbUSTimer(IN := FALSE);

									eGotoOpsStep	:= InvertStepUSStandby;
								END_IF

							END_IF

					END_CASE

				InvertStepEntToEnd:
					CASE p_eUSCommMod OF
						McSetCommModSMEMA:
							IF p_bUSSMEMATransporting = FALSE AND bUSTimerRun = FALSE THEN
								eConvAct	:= ConvActStop;

								IF p_eConvStatus = Done AND p_eConvStat = ConvActStop THEN
									eConvAct		:= ConvActIdle;

									eGotoOpsStep	:= InvertStepUSStandby;

									bPaused	:= p_bStop OR p_bStep;

								END_IF

							ELSE
								IF p_bUSSMEMAConvStart OR bUSTimerRun THEN
									sStepTxt	:= 'Conveyor Entering Board';
									eConvAct	:= ConvActEnt;
								END_IF

								IF (p_bConvHvBrd = TRUE) OR bUSTimerRun THEN
									bHvBrd := TRUE;
								END_IF

								IF p_bUSSMEMAConvStop AND bUSTimerRun = FALSE THEN
									sStepTxt	:= 'Conveyor Stopping';
									eConvAct	:= ConvActStop;
								END_IF

								//Waiting Conveyor Reach End for Invert Mode
								IF p_usiLinkProdRcpCurrRcpMcMod = 0 THEN

									IF (p_eUSSMEMAStatus = Done AND p_eUSSMEMAStat = SMEMAActRun) OR (bUSTimerRun = TRUE) THEN
										eUSSMEMAAct		:= SMEMAActIdle;
										eGotoOpsStep	:= InvertStepInvertComplChk;

										IF p_eConvStatus <> Busy THEN
											bPaused	:= p_bStop OR p_bStep;
										END_IF
									END_IF

								ELSIF p_usiLinkProdRcpCurrRcpMcMod = 1 THEN
									IF ((p_eUSSMEMAStatus = Done AND p_eUSSMEMAStat = SMEMAActRun) OR (bUSTimerRun = TRUE)) AND p_eConvStatus = Done AND p_eConvStat = ConvActEnt THEN
										eUSSMEMAAct		:= SMEMAActIdle;
										eGotoOpsStep	:= InvertStepInvertComplChk;

										IF p_eConvStatus <> Busy THEN
											bPaused	:= p_bStop OR p_bStep;
										END_IF
									END_IF

								END_IF

							END_IF

						McSetCommModHermes:
							IF p_bUSHermesTransporting OR bUSTimerRun = TRUE THEN
								sStepTxt	:= 'Conveyor Entering Board';
								eConvAct	:= ConvActEnt;
							END_IF

							IF p_bUSHermesStopTransport = TRUE  AND bUSTimerRun = FALSE THEN
								sStepTxt	:= 'Conveyor Stopping';
								eConvAct	:= ConvActStop;
							END_IF

							IF (p_bConvHvBrd = TRUE) OR (bUSTimerRun = TRUE) THEN
								bHvBrd := TRUE;
							END_IF

							//Waiting Conveyor Reach End for Invert Mode
							IF p_usiLinkProdRcpCurrRcpMcMod = 0 THEN

								IF (p_bUSHermesTransporting = FALSE) OR (bUSTimerRun) THEN
									IF p_eConvStat = ConvActStop THEN
										IF p_eConvStatus = Done THEN
											eConvAct		:= ConvActIdle;
											eGotoOpsStep	:= InvertStepUSStandby;
										END_IF
									ELSE
										eGotoOpsStep	:= InvertStepInvertComplChk;
									END_IF

									IF p_eConvStatus <> Busy THEN
										bPaused	:= p_bStop OR p_bStep;
									END_IF
								END_IF

							ELSIF p_usiLinkProdRcpCurrRcpMcMod = 1 THEN

								IF ((p_bUSHermesTransporting = FALSE ) OR (bUSTimerRun)) THEN
									IF p_eConvStat = ConvActStop THEN
										IF p_eConvStatus = Done THEN
											eConvAct		:= ConvActIdle;
											eGotoOpsStep	:= InvertStepUSStandby;
										END_IF
									ELSE
										IF p_eConvStatus = Done AND p_eConvStat = ConvActEnt THEN
											eGotoOpsStep	:= InvertStepInvertComplChk;
										END_IF
									END_IF

									IF p_eConvStatus <> Busy THEN
										bPaused	:= p_bStop OR p_bStep;
									END_IF
								END_IF

							END_IF

					END_CASE

				InvertStepEntToInOff:
					CASE p_eUSCommMod OF
						McSetCommModSMEMA:
							IF p_bUSSMEMATransporting = FALSE AND bUSTimerRun = FALSE THEN
								eConvAct	:= ConvActStop;

								IF p_eConvStatus = Done AND p_eConvStat = ConvActStop THEN
									eConvAct		:= ConvActIdle;
									eGotoOpsStep	:= InvertStepUSStandby;

									bPaused	:= p_bStop OR p_bStep;

								END_IF

							ELSE
								IF p_bUSSMEMAConvStart OR bUSTimerRun THEN
									sStepTxt	:= 'Conveyor Entering Board';
									eConvAct	:= ConvActEntToInOff;
								END_IF

								IF (p_bConvHvBrd = TRUE) OR (bUSTimerRun = TRUE) THEN
									bHvBrd := TRUE;
								END_IF

								IF p_bUSSMEMAConvStop AND bUSTimerRun = FALSE THEN
									sStepTxt	:= 'Conveyor Stopping';
									eConvAct	:= ConvActStop;
								END_IF

								IF ((p_eUSSMEMAStatus = Done AND p_eUSSMEMAStat = SMEMAActRun) OR (bUSTimerRun = TRUE)) AND p_eConvStatus = Done AND p_eConvStat = ConvActEntToInOff THEN
									eUSSMEMAAct		:= SMEMAActIdle;
									eGotoOpsStep	:= InvertStepStopperBlkAftEnt;

									IF p_eConvStatus <> Busy THEN
										bPaused	:= p_bStop OR p_bStep;
									END_IF
								END_IF

							END_IF

						McSetCommModHermes:
							IF p_bUSHermesTransporting OR bUSTimerRun = TRUE THEN
								sStepTxt	:= 'Conveyor Entering Board';
								eConvAct	:= ConvActEntToInOff;
							END_IF

							IF p_bUSHermesStopTransport = TRUE AND bUSTimerRun = FALSE THEN
								sStepTxt	:= 'Conveyor Stopping';
								eConvAct	:= ConvActStop;
							END_IF

							IF (p_bConvHvBrd = TRUE) OR (bUSTimerRun = TRUE) THEN
								bHvBrd	:= TRUE;
							END_IF

							IF ((p_bUSHermesTransporting = FALSE) OR (bUSTimerRun)) THEN
								IF p_eConvStat = ConvActStop THEN
									IF p_eConvStatus = Done THEN
										eConvAct		:= ConvActIdle;
										eGotoOpsStep	:= InvertStepUSStandby;
									END_IF
								ELSE
									IF p_eConvStatus = Done AND p_eConvStat = ConvActEntToInOff THEN
										eGotoOpsStep	:= InvertStepStopperBlkAftEnt;
									END_IF
								END_IF

								IF p_eConvStatus <> Busy THEN
									bPaused	:= p_bStop OR p_bStep;
								END_IF
							END_IF

					END_CASE

				InvertStepStopperBlkAftEnt:
					sStepTxt	:= 'Stopper Block After Entering Board';

					eStopperAct	:= PneuActExt;

					IF p_eStopperStatus = Done AND p_eStopperStat = PneuActExt THEN
						eStopperAct		:= PneuActIdle;
						eGotoOpsStep	:= InvertStepRev;

						bPaused	:= p_bStop OR p_bStep;
					END_IF

				InvertStepRev:
					sStepTxt	:= 'Conveyor Reverse Board';

					eConvAct	:= ConvActRevImmedStart;

					IF p_eConvStatus = Done AND p_eConvStat = ConvActRevImmedStart THEN
						eConvAct		:= ConvActIdle;

						eGotoOpsStep	:= InvertStepInvertComplChk;

						bPaused	:= p_bStop OR p_bStep;
					END_IF

				InvertStepInvertComplChk:
					sStepTxt		:= 'Checking Invert Complete Condition';

					IF eInvertCurrPos <> eInvertReqPos THEN
						IF p_bClampPrep AND p_bClampDis=FALSE THEN
							eGotoOpsStep	:= InvertStepClampBlkBefInvert;
						ELSE
							IF (p_bInletShutterPrep AND p_bInletShutterDis=FALSE) OR (p_bOutletShutterPrep AND p_bOutletShutterDis=FALSE) THEN
								eGotoOpsStep	:= InvertStepShuttersCloseBefInvert;
							ELSE
								eGotoOpsStep	:= InvertStepInvert;
							END_IF
						END_IF
					ELSE
						IF (p_bInletShutterPrep AND p_bInletShutterDis=FALSE) OR (p_bOutletShutterPrep AND p_bOutletShutterDis=FALSE) THEN
							IF p_bOutletShutterOpen THEN
								eGotoOpsStep	:= InvertStepDSStandby;
							ELSE
								eGotoOpsStep	:= InvertStepOutletShutterOpen;
							END_IF
						ELSE
							eGotoOpsStep	:= InvertStepDSStandby;
						END_IF
					END_IF

					IF p_eConvStatus <> Busy THEN
						bPaused	:= p_bStop OR p_bStep;
					END_IF

				InvertStepClampBlkBefInvert:
					sStepTxt	:= 'Clamp Block Prior to Inversion';

					eClampAct	:= PneuActExt;

					IF p_eClampStatus = Done AND p_eClampStat = PneuActExt THEN

						eClampAct		:= PneuActIdle;

						IF (p_bInletShutterPrep AND p_bInletShutterDis=FALSE) OR (p_bOutletShutterPrep AND p_bOutletShutterDis=FALSE) THEN
							eGotoOpsStep	:= InvertStepShuttersCloseBefInvert;
						ELSE
							eGotoOpsStep	:= InvertStepInvert;
						END_IF

						bPaused	:= p_bStop OR p_bStep;
					END_IF

				InvertStepShuttersCloseBefInvert:
					sStepTxt			:= 'Closing Shutters Prior to Inversion';

					eInletShutterAct	:= PneuActExt;
					eOutletShutterAct	:= PneuActExt;

					IF (p_eInletShutterStatus = Done AND p_eInletShutterStat = PneuActExt) AND (p_eOutletShutterStatus = Done AND p_eOutletShutterStat = PneuActExt) THEN

						eInletShutterAct	:= PneuActIdle;
						eOutletShutterAct	:= PneuActIdle;

						eGotoOpsStep	:= InvertStepInvert;

						bPaused	:= p_bStop OR p_bStep;
					END_IF

				InvertStepInvert:
					sStepTxt	:= 'Inverter Turning';

					IF eInvertReqPos = InvertCurrPosAtRemote THEN
						eInvertAct	:= MotorBrkActCW;
					ELSIF eInvertReqPos = InvertCurrPosAtHome THEN
						eInvertAct	:= MotorBrkActCCW;
					END_IF

					IF p_eInvertStatus = Done AND (p_eInvertStat = MotorBrkActCW OR p_eInvertStat = MotorBrkActCCW)THEN
						eInvertAct		:= MotorBrkActIdle;

						IF (p_bClampPrep AND p_bClampDis=FALSE) OR bClampDisInitUnblk THEN

							bClampDisInitUnblk	:= FALSE;

							eGotoOpsStep	:= InvertStepClampUnblkAftInvert;

						ELSE
							IF eInvertCurrPos = InvertCurrPosAtRemote THEN

								IF bInvertPosInvalidSkipInit THEN
									eGotoOpsStep	:= InvertStepInvalidPosRecoverBrd;
								ELSE
									IF p_bLeftSen = TRUE THEN
										eGotoOpsStep	:= InvertStepPreExit;
									ELSE
										eGotoOpsStep	:= InvertStepChkCondition;
									END_IF
								END_IF

							ELSIF eInvertCurrPos = InvertCurrPosAtHome THEN

								IF bInvertPosInvalidSkipInit THEN
									eGotoOpsStep	:= InvertStepInvalidPosRecoverBrd;
								ELSE
									IF p_bRightSen = TRUE THEN
										eGotoOpsStep	:= InvertStepStopperUnblkAftInvert;
									ELSE
										eGotoOpsStep	:= InvertStepChkCondition;
									END_IF
								END_IF
							END_IF
						END_IF

						bPaused	:= p_bStop OR p_bStep;
					END_IF

				InvertStepClampUnblkAftInvert:
					sStepTxt	:= 'Clamp Unblock After Invert';

					eClampAct	:= PneuActRet;

					IF p_eClampStatus = Done AND p_eClampStat = PneuActRet THEN
						eClampAct		:= PneuActIdle;

						IF eInvertCurrPos = InvertCurrPosAtRemote THEN

							IF bInvertPosInvalidSkipInit THEN
								eGotoOpsStep	:= InvertStepInvalidPosRecoverBrd;
							ELSE
								IF p_bLeftSen = TRUE THEN
									eGotoOpsStep	:= InvertStepPreExit;
								ELSE
									eGotoOpsStep	:= InvertStepChkCondition;
								END_IF
							END_IF

						ELSIF eInvertCurrPos = InvertCurrPosAtHome THEN

							IF bInvertPosInvalidSkipInit THEN
								eGotoOpsStep	:= InvertStepInvalidPosRecoverBrd;
							ELSE
								IF p_bRightSen = TRUE THEN
									eGotoOpsStep	:= InvertStepStopperUnblkAftInvert;
								ELSE
									eGotoOpsStep	:= InvertStepChkCondition;
								END_IF
							END_IF
						END_IF

						bPaused	:= p_bStop OR p_bStep;

					END_IF

				InvertStepInvalidPosRecoverBrd:
					sStepTxt		:= 'Conveyor Recovering Board Status';

					eConvAct	:= ConvActInit;

					IF p_eConvStatus = Done AND p_eConvStat = ConvActInit THEN
						eConvAct		:= ConvActIdle;

						IF p_bRightSen = TRUE THEN
							bHvBrd := TRUE;
							bGdBrd			:= p_bInitGdBrd;

							bInvertPosInvalidSkipInit := FALSE;

							IF eInvertCurrPos = InvertCurrPosAtRemote THEN
								IF (p_bInletShutterPrep AND p_bInletShutterDis=FALSE) OR (p_bOutletShutterPrep AND p_bOutletShutterDis=FALSE) THEN
									IF p_bOutletShutterOpen THEN
										eGotoOpsStep	:= InvertStepDSStandby;
									ELSE
										eGotoOpsStep	:= InvertStepOutletShutterOpen;
									END_IF
								ELSE
									eGotoOpsStep	:= InvertStepDSStandby;
								END_IF
							ELSIF eInvertCurrPos = InvertCurrPosAtHome THEN
								eGotoOpsStep	:= InvertStepStopperUnblkAftInvert;
							END_IF

						ELSE
							bInvertPosInvalidSkipInit := FALSE;
							eGotoOpsStep	:= InvertStepChkCondition;
						END_IF

						bPaused	:= p_bStop OR p_bStep;
					END_IF

				InvertStepStopperUnblkAftInvert:
					sStepTxt	:= 'Stopper Unblock After Invert';

					eStopperAct	:= PneuActRet;

					IF p_eStopperStatus = Done AND p_eStopperStat = PneuActRet THEN
						eStopperAct		:= PneuActIdle;

						IF (p_bInletShutterPrep AND p_bInletShutterDis=FALSE) OR (p_bOutletShutterPrep AND p_bOutletShutterDis=FALSE) THEN
							IF p_bOutletShutterOpen THEN
								eGotoOpsStep	:= InvertStepDSStandby;
							ELSE
								eGotoOpsStep	:= InvertStepOutletShutterOpen;
							END_IF
						ELSE
							eGotoOpsStep	:= InvertStepDSStandby;
						END_IF

						bPaused	:= p_bStop OR p_bStep;
					END_IF

				InvertStepPreExit:
					sStepTxt		:= 'Conveyor Pre-Exiting Board';

					eConvAct	:= ConvActPreExit;

					IF p_eConvStatus = Done AND p_eConvStat = ConvActPreExit THEN
						eConvAct		:= ConvActIdle;

						IF (p_bInletShutterPrep AND p_bInletShutterDis=FALSE) OR (p_bOutletShutterPrep AND p_bOutletShutterDis=FALSE) THEN
							IF p_bOutletShutterOpen THEN
								eGotoOpsStep	:= InvertStepDSStandby;
							ELSE
								eGotoOpsStep	:= InvertStepOutletShutterOpen;
							END_IF
						ELSE
							eGotoOpsStep	:= InvertStepDSStandby;
						END_IF

						bPaused	:= p_bStop OR p_bStep;
					END_IF

				InvertStepDSInOutletShutterOpen:
					sStepTxt	:= 'DS: Opening Inlet & Outlet Shutter';

					eInletShutterAct	:= PneuActRet;
					eOutletShutterAct	:= PneuActRet;

					IF (p_eInletShutterStatus = Done AND p_eInletShutterStat = PneuActRet)
						AND (p_eOutletShutterStatus = Done AND p_eOutletShutterStat = PneuActRet)THEN

						eInletShutterAct	:= PneuActIdle;
						eOutletShutterAct	:= PneuActIdle;

						eGotoOpsStep	:= InvertStepDSStandby;

						bPaused	:= p_bStop OR p_bStep;
					END_IF

				InvertStepOutletShutterOpen:
					sStepTxt	:= 'Opening Outlet Shutter';

					eOutletShutterAct	:= PneuActRet;

					IF p_eOutletShutterStatus = Done AND p_eOutletShutterStat = PneuActRet THEN
						eOutletShutterAct	:= PneuActIdle;

						eGotoOpsStep	:= InvertStepDSStandby;

						bPaused	:= p_bStop OR p_bStep;
					END_IF

				InvertStepDSStandby:
					sStepTxt	:= 'In Downstream Standby Condition';

					bDSTimerRun	:= FALSE;

					IF p_eConvDirection = ConvDirLToL OR p_eConvDirection = ConvDirRToL THEN
						bConvSen	:= p_bLeftSen;
					ELSE
						bConvSen	:= p_bRightSen;
					END_IF

					IF bConvSen = TRUE OR p_eConvStatus <> Busy THEN
						bReachedEnd	:= TRUE;
					END_IF

					IF p_bDBAOnRgtSen THEN
						IF p_bDSAllow = TRUE AND bReachedEnd = TRUE THEN
							bReachedEnd		:= FALSE;
							eGotoOpsStep	:= InvertStepDSCommTmr;
						ELSIF (bReachedEnd = TRUE) AND (bConvSen = FALSE) THEN
							bReachedEnd		:= FALSE;
							eGotoOpsStep	:= InvertStepDSTmr;
						END_IF
					ELSE
						IF p_bDSAllow = TRUE THEN
							bReachedEnd		:= FALSE;
							eGotoOpsStep	:= InvertStepDSCommTmr;
						ELSIF (bReachedEnd = TRUE) AND (bConvSen = FALSE) THEN
							bReachedEnd		:= FALSE;
							eGotoOpsStep	:= InvertStepDSTmr;
						END_IF
					END_IF

					IF p_eConvStatus <> Busy THEN
						bPaused	:= p_bStop OR p_bStep;
					END_IF

				InvertStepDSTmr:
					sStepTxt	:= 'Removing Board By Timer';

					IF p_eConvDirection = ConvDirLToL OR p_eConvDirection = ConvDirRToL THEN
						bConvSen	:= p_bLeftSen;
					ELSE
						bConvSen	:= p_bRightSen;
					END_IF

					fbDSTimer(IN := NOT bConvSen);

					IF fbDSTimer.Q = TRUE THEN
						bDSTimerRun		:= TRUE;
						fbDSTimer(IN := FALSE);

						bHvBrd := FALSE;

						eConvAct		:= ConvActIdle;

						eGotoOpsStep	:= InvertStepChkCondition;

					ELSIF bConvSen = TRUE THEN
						bDSTimerRun		:= FALSE;
						fbDSTimer(IN := FALSE);

						eGotoOpsStep	:= InvertStepDSStandby;

					ELSE
						IF p_eConvStatus <> Busy THEN
							bPaused	:= p_bStop;

							IF bPaused = TRUE THEN
								bDSTimerRun	:= FALSE;
								fbDSTimer(IN := FALSE);
							END_IF
						END_IF

					END_IF

				InvertStepDSCommTmr:
					sStepTxt	:= 'Communicating Downstream Machine';

					IF p_eConvDirection = ConvDirLToL OR p_eConvDirection = ConvDirRToL THEN
						IF p_bLeftSen = TRUE OR p_eConvStatus <> Busy THEN
							bReachedEnd	:= TRUE;
						END_IF

						IF bReachedEnd = TRUE THEN
							fbDSTimer(IN := NOT p_bLeftSen);
						END_IF
					ELSE
						IF p_bRightSen = TRUE OR p_eConvStatus <> Busy THEN
							bReachedEnd	:= TRUE;
						END_IF

						IF bReachedEnd = TRUE THEN
							fbDSTimer(IN := NOT p_bRightSen);
						END_IF
					END_IF

					CASE p_eDSCommMod OF
						McSetCommModSMEMA:
							eDSSMEMAAct	:= SMEMAActRun;

							IF p_bDSSMEMAConvStart = TRUE THEN
								bDSTimerRun	:= FALSE;
								fbDSTimer(IN := FALSE);

								bReachedEnd	:= FALSE;

								eGotoOpsStep	:= InvertStepExitBrd;

							ELSIF fbDSTimer.Q = TRUE THEN
								bDSTimerRun		:= TRUE;
								fbDSTimer(IN := FALSE);
								bHvBrd := FALSE;

								bReachedEnd		:= FALSE;
								eDSSMEMAAct		:= SMEMAActIdle;
								eConvAct		:= ConvActIdle;

								eGotoOpsStep	:= InvertStepChkCondition;

							ELSIF p_bDSAllow = FALSE THEN
								bDSTimerRun		:= FALSE;
								fbDSTimer(IN := FALSE);

								bReachedEnd		:= FALSE;
								eDSSMEMAAct		:= SMEMAActIdle;
								eConvAct		:= ConvActIdle;

								eGotoOpsStep	:= InvertStepDSStandby;

							ELSE
								IF p_eConvStatus <> Busy THEN
									bPaused	:= p_bStop;

									IF bPaused = TRUE THEN
										fbDSTimer(IN := FALSE);

										eDSSMEMAAct	:= SMEMAActIdle;
									END_IF
								END_IF

							END_IF

						McSetCommModHermes:
							IF p_bDSHermesTransporting = TRUE THEN
								bDSTimerRun	:= FALSE;
								fbDSTimer(IN := FALSE);

								bReachedEnd	:= FALSE;

								eGotoOpsStep	:= InvertStepExitBrd;

							ELSIF fbDSTimer.Q = TRUE THEN
								bDSTimerRun	:= TRUE;
								fbDSTimer(IN := FALSE);
								bHvBrd := FALSE;

								bReachedEnd	:= FALSE;
								eConvAct		:= ConvActIdle;

								eGotoOpsStep	:= InvertStepChkCondition;

							ELSIF p_bDSAllow = FALSE THEN
								bDSTimerRun	:= FALSE;
								fbDSTimer(IN := FALSE);

								bReachedEnd	:= FALSE;

								eGotoOpsStep	:= InvertStepDSStandby;

							ELSE
								IF p_eConvStatus <> Busy THEN
									bPaused	:= p_bStop;

									IF bPaused = TRUE THEN
										fbDSTimer(IN := FALSE);
									END_IF
								END_IF

							END_IF

					END_CASE

				InvertStepExitBrd:
					CASE p_eDSCommMod OF
						McSetCommModSMEMA:
							eConvAct	:= ConvActExit;

							IF ((p_eDSSMEMAStatus = Done AND p_eDSSMEMAStat = SMEMAActRun) OR (bDSTimerRun)) AND (p_eConvStatus = Done AND p_eConvStat = ConvActExit) THEN

								eDSSMEMAAct		:= SMEMAActIdle;
								eConvAct		:= ConvActIdle;

								bHvBrd := FALSE;
								p_bConvHvBrd := FALSE;
								eGotoOpsStep	:= InvertStepChkCondition;

								bPaused	:= p_bStop OR p_bStep;

							END_IF

						McSetCommModHermes:
							eConvAct := ConvActExit;

							IF ((p_bDSHermesTransporting = FALSE) OR (bDSTimerRun)) AND (p_eConvStatus = Done AND p_eConvStat = ConvActExit) THEN
								eConvAct := ConvActIdle;

								bHvBrd := FALSE;
								p_bConvHvBrd := FALSE;

								eGotoOpsStep := InvertStepChkCondition;

								bPaused := p_bStop OR p_bStep;
							END_IF

					END_CASE

			END_CASE

		END_IF

	END_IF

	//Board Inserted/Removed
	bBrdInserted		:= bUSTimerRun;
	bBrdRemoved			:= bDSTimerRun;

	//Operation Step Status
	IF (eOpsStep = InvertStepInitConvAwayLftSen) OR (eOpsStep = InvertStepInitConvAwayRgtSen) OR (eOpsStep = InvertStepInitConvTwdLftSen) OR (eOpsStep = InvertStepInitConvTwdRgtSen) OR (eOpsStep = InvertStepInitConvToRgt) THEN
		bStepInitConv	:= TRUE;
	ELSE
		bStepInitConv	:= FALSE;
	END_IF

	bStepInitAwayStopper		:= (eOpsStep = InvertStepInitConvAwayLftSen) OR (eOpsStep = InvertStepInitConvAwayRgtSen);
	bStepInitTwdStopper			:= (eOpsStep = InvertStepInitConvTwdLftSen) OR (eOpsStep = InvertStepInitConvTwdRgtSen);
	bStepInitDone				:= (eOpsStep > InvertStepInitShuttersInOutClose) AND bInvertPosInvalidSkipInit=FALSE;
	bStepUSStandby				:= eOpsStep = InvertStepUSStandby;
	bStepUSCommTmr				:= eOpsStep = InvertStepUSCommTmr;
	bStepEntToEnd				:= eOpsStep = InvertStepEntToEnd;
	bStepEntToInOff				:= eOpsStep = InvertStepEntToInOff;
	bStepRev					:= eOpsStep = InvertStepRev;
	bStepPreExit				:= eOpsStep = InvertStepPreExit;
	bStepDSStandby				:= eOpsStep = InvertStepDSStandby;
	bStepDSCommTmr				:= eOpsStep = InvertStepDSCommTmr;
	bStepExitBrd				:= eOpsStep = InvertStepExitBrd;
	bStepInvert					:= eOpsStep = InvertStepInvert;
	bStepAWMov					:= eOpsStep = InvertStepAWMov;
END_ACTION
```
